// TwinCAT 3 PLC project TcKNXnetIP_Tunneling_Lib
// Title: TcKNXnetIP_Tunneling_Lib
// Company: Gauggel
// Author: Gauggel Alexander
// ProjectVersion: 1.0.0
// Description: Library for KNXnetIP Tunnelling connection (write/read group addresses) License: MIT License Disclaimer: This software is provided "as is", without warranty of any kind, express or implied. The author shall not be held liable for any damages arising from the use of this software.
// ProgramVersion: 3.1.4026.20
// libraries:
//   Tc2_Standard, * (Beckhoff Automation GmbH)
//   Tc2_System, * (Beckhoff Automation GmbH)
//   Tc2_TcpIp, * (Beckhoff Automation GmbH)
// project tree:
//   KNXnetIPTunnelingServer/DUTs/ E_KNXnetIP_COMMON_CONSTANTS.TcDUT, E_KNXnetIP_COMMON_ERROR.TcDUT, E_KNXnetIP_CONNECTIONSTATE_RESPONSE_ERROR.TcDUT, E_KNXnetIP_CONNECTION_TYPE.TcDUT, E_KNXnetIP_CONNECT_RESPONSE_ERROR.TcDUT, E_KNXnetIP_CORE.TcDUT, E_KNXnetIP_DEVICE_MANAGEMENT.TcDUT, E_KNXnetIP_ROUTING.TcDUT, E_KNXnetIP_ServiceTypes.TcDUT, E_KNXnetIP_TUNNELING.TcDUT, E_KNXnetIP_TUNNELING_CONNECT_ERROR.TcDUT, ST_KNXnetIP_cEMI.TcDUT, ST_KNXnetIP_CommonHeader.TcDUT, ST_KNXnetIP_ConnectionHeader.TcDUT, ST_KNXnetIP_ConnectionStateResponse.TcDUT, ST_KNXnetIP_ConnectResponse.TcDUT, ST_KNXnetIP_DisconnectRequest.TcDUT, ST_KNXnetIP_DisconnectResponse.TcDUT, ST_KNXnetIP_Message.TcDUT, ST_KNXnetIP_MessageOfAllGroupAddresses.TcDUT, ST_KNXnetIP_Message_Buffer.TcDUT, ST_KNX_GroupAddress.TcDUT, ST_KNX_PhysicalAddress.TcDUT
//   KNXnetIPTunnelingServer/DUTs/Interpreter/ ST_KNX_DPT_B2.TcDUT, ST_KNX_DPT_ControlDimming.TcDUT
//   KNXnetIPTunnelingServer/DUTs/StateMachines/ E_KNXnetIPStateConnection.TcDUT, E_KNXnetIPStateReceivedTelegrams.TcDUT, E_KNXnetIPStateRequest.TcDUT, E_KNXnetIPStateTransmitTelegrams.TcDUT
//   KNXnetIPTunnelingServer/ITFs/ I_KNXnetIP_Tunneling.TcIO, I_KNX_DPT_Builder.TcIO, I_KNX_DPT_Interpreter.TcIO
//   KNXnetIPTunnelingServer/PARAMs/ KNXnetIP_TIMEOUT_CONSTANS.TcGVL
//   KNXnetIPTunnelingServer/POUs/ F_KNX_GROUPADDRESS_TO_WORD.TcPOU, F_KNX_PHYSICALADDRESS_TO_WORD.TcPOU, F_WORD_TO_KNX_GROUPADDRESS.TcPOU, F_WORD_TO_KNX_PHYSICALADDRESS.TcPOU, KNXnetIPTunnelingServer.TcPOU, KNXnetIP_Message_FiFoBuffer.TcPOU, KNX_DatapointTypes_Builder.TcPOU, KNX_DatapointTypes_Interpreter.TcPOU
//   KNXnetIP_Devices/Button/ FB_KNXnetIP_Button.TcPOU
//   KNXnetIP_Devices/ FB_KNXnetIP_Device_Abstract.TcPOU
//   KNXnetIP_Devices/Light/ FB_KNXnetIP_Light.TcPOU
//   Project Information/ F_GetCompany.TcPOU, F_GetTitle.TcPOU, F_GetVersion.TcPOU
//   Version/ Global_Version.TcGVL

// ---- KNXnetIPTunnelingServer/DUTs/E_KNXnetIP_COMMON_CONSTANTS.TcDUT
{attribute 'qualified_only'}
{attribute 'to_string'}
TYPE E_KNXnetIP_COMMON_CONSTANTS :
(
	KNXNETIP_VERSION_10 := 16#10,			// Identifier for KNXnet/IP protocol version 1.0
	HEADER_SIZE_10		:= 16#06			// constant size of KNXnet/IP header as defined in protocol version 1.0
) BYTE
;
END_TYPE

// ---- KNXnetIPTunnelingServer/DUTs/E_KNXnetIP_COMMON_ERROR.TcDUT
{attribute 'qualified_only'}
{attribute 'to_string'}
TYPE E_KNXnetIP_COMMON_ERROR :
(
	E_NO_ERROR 					:= 16#00,			// Operation successful
	E_HOST_PROTOCOL_TYPE 		:= 16#01,			// The requested host protocol is not supported by the KNXnet/IP device.
	E_VERSION_NOT_SUPPORTED		:= 16#02,			// The requested protocol version is not supported by the KNXnet/IP device.
	E_SEQUENCE_NUMBER	 		:= 16#04,			// The received sequence number is out of order.
	E_ERROR 					:= 16#0F			// Any further undefined, possibly implementation specific error has occurred.
) BYTE 
;
END_TYPE

// ---- KNXnetIPTunnelingServer/DUTs/E_KNXnetIP_CONNECTIONSTATE_RESPONSE_ERROR.TcDUT
{attribute 'qualified_only'}
{attribute 'to_string'}
TYPE E_KNXnetIP_CONNECTIONSTATE_RESPONSE_ERROR :
(
	E_NO_ERROR 					:= 16#00,		// The connection state is normal.
	E_CONNECTION_ID 			:= 16#21,		// The KNXnet/IP Server device cannot find an active data connection with the specified ID.
	E_DATA_CONNECTION 			:= 16#26,		// The KNXnet/IP Server device detects an error concerning the data connection with the specified ID.
	E_KNX_CONNECTION 			:= 16#27		// The KNXnet/IP Server device detects an error concerning the KNX connection with the specified ID.
) BYTE 
;
END_TYPE

// ---- KNXnetIPTunnelingServer/DUTs/E_KNXnetIP_CONNECTION_TYPE.TcDUT
{attribute 'qualified_only'}
{attribute 'to_string'}
TYPE E_KNXnetIP_CONNECTION_TYPE :
(
	DEVICE_MGMT_CONNECTION		:= 16#03,			// Data connection used to configure a KNXnet/IP device.
	TUNNEL_CONNECTION			:= 16#04,			// Data connection used to forward KNX telegrams between two KNXnet/IP devices.
	REMLOG_CONNECTION			:= 16#06,			// Data connection used for configuration and data transfer with a remote logging server.
	REMCONF_CONNECTION			:= 16#07,			// Data connection used for data transfer with a remote configuration server.
	OBJSVR_CONNECTION			:= 16#08			// Data connection used for configuration and data transfer with an Object Server in a KNXnet/IP device. 
) BYTE
;
END_TYPE

// ---- KNXnetIPTunnelingServer/DUTs/E_KNXnetIP_CONNECT_RESPONSE_ERROR.TcDUT
{attribute 'qualified_only'}
{attribute 'to_string'}
TYPE E_KNXnetIP_CONNECT_RESPONSE_ERROR :
(
	E_NO_ERROR 						:= 16#00,		// The connection is established successfully.
	E_CONNECTION_TYPE 				:= 16#22,		// The KNXnet/IP Server device does not support the requested connection type.
	E_CONNECTION_OPTION 			:= 16#23,		// The KNXnet/IP Server device does not support one or more requested connection options.
	E_NO_MORE_CONNECTIONS 			:= 16#24,		// The KNXnet/IP Server device cannot accept the new data connection because its maximum amount of concurrent connections is already used.
	E_AUTHORISATION_ERROR 			:= 16#28,		// The Client is not authorised to establish the requested connection The Client is not authorised to use the requested IA in the Extended CRI.
	E_NO_TUNNELING_ADDRESS 			:= 16#2D,		// The IA requested in the Extended CRI is not a Tunnelling IA.
	E_CONNECTION_IN_USE 			:= 16#2E		// The IA requested for this connection is in use. 
) BYTE
;
END_TYPE

// ---- KNXnetIPTunnelingServer/DUTs/E_KNXnetIP_CORE.TcDUT
{attribute 'qualified_only'}
{attribute 'to_string'}
TYPE E_KNXnetIP_CORE :
(
	SEARCH_REQUEST 				:= 16#0201,		// Sent by KNXnet/IP Client to search available KNXnet/IP Servers
	SEARCH_RESPONSE				:= 16#0202,		// Sent by KNXnet/IP Server when receiving a KNXnet/IP SEARCH_REQUEST
	DESCRIPITON_REQUEST			:= 16#0203,		// Sent by KNXnet/IP Client to a KNXnet/IP Server to retrieve information about capabilities and supported services
	DESCRIPTION_RESPONSE		:= 16#0204,		// Sent by KNXnet/IP Server in response to a DESCRIPTION_REQUEST to provide information about the server implementation
	CONNECT_REQUEST				:= 16#0205,		// Sent by KNXnet/IP Client for establishing a communication channel to a KNXnet/IP Server.
	CONNECT_RESPONSE			:= 16#0206,		// Sent by KNXnet/IP Server as answer to CONNECT_REQUEST telegram.
	CONNECTIONSTATE_REQUEST		:= 16#0207,		// Sent by KNXnet/IP Client for requesting the connection state of an established connection to a KNXnet/IP Server.
	CONNECTIONSTATE_RESPONSE	:= 16#0208,		// Sent by KNXnet/IP Server when receiving a CONNECTIONSTATE_REQUEST for an established connection.
	DISCONNECT_REQUEST			:= 16#0209,		// Sent by KNXnet/IP device, typically the KNXnet/IP Client, to terminate an established connection.
	DISCONNECT_RESPONSE			:= 16#020A,		// Sent by KNXnet/IP device, typically the KNXnet/IP Server, in response to a DISCONNECT_REQUEST.
	SECURE_WRAPPER				:= 16#0950,		// Contains an encrypted frame plus data for ensuring data integrity and freshness.
	SESSION_REQUEST				:= 16#0951,		// Used to initiate the secure connection setup handshake for a new secure communication session.
	SESSION_RESPONSE			:= 16#0952,		// Sent in response to a received secure session request frame.
	SESSION_AUTHENTICATE		:= 16#0953,		// Sent after the Diffie-Hellman handshake to authenticate the user against the server.
	SESSION_STATUS				:= 16#0954,		// Sent in any stage of the secure session handshake to indicate an error condition or status information.
	TIMER_NOTIFY				:= 16#0955		// Used to ensure synchronization of the multicast group member's timer values.
) WORD 
;
END_TYPE

// ---- KNXnetIPTunnelingServer/DUTs/E_KNXnetIP_DEVICE_MANAGEMENT.TcDUT
{attribute 'qualified_only'}
{attribute 'to_string'}
TYPE E_KNXnetIP_DEVICE_MANAGEMENT :
(
	DEVICE_CONFIGURATION_REQUEST	:= 16#0310,			// Reads/Writes KNXnet/IP device configuration data (Interface Object Properties)
	DEVICE_CONFIGURATION_ACK		:= 16#0311			// Sent by a KNXnet/IP device to confirm the reception of the DEVICE_CONFIGURATION_REQUEST. 
) WORD 
;
END_TYPE

// ---- KNXnetIPTunnelingServer/DUTs/E_KNXnetIP_ROUTING.TcDUT
{attribute 'qualified_only'}
{attribute 'to_string'}
TYPE E_KNXnetIP_ROUTING :
(
	ROUTING_INDICATION 		:= 16#0530,		// Used for sending KNX telegrams over IP networks. This service is unconfirmed.
	ROUTING_LOST_MESSAGE	:= 16#0531		// Used for indication of lost KNXnet/IP Routing messages. This service is unconfirmed.
) WORD
;
END_TYPE

// ---- KNXnetIPTunnelingServer/DUTs/E_KNXnetIP_ServiceTypes.TcDUT
{attribute 'qualified_only'}
{attribute 'to_string'}
TYPE E_KNXnetIP_ServiceTypes :
(
	eL_DataReq		 	:= 16#11,
	eL_DataCon			:= 16#2E,
	eL_DataInd			:= 16#29
)BYTE
;
END_TYPE

// ---- KNXnetIPTunnelingServer/DUTs/E_KNXnetIP_TUNNELING.TcDUT
{attribute 'qualified_only'}
{attribute 'to_string'}
TYPE E_KNXnetIP_TUNNELING :
(
	TUNNELING_REQUEST 	:= 16#0420,		// Used for sending and receiving single KNX telegrams between KNXnet/IP Client and - Server.
	TUNNELING_ACK		:= 16#0421		// Sent by a KNXnet/IP device to confirm the reception of the TUNNELING_REQUEST.
) WORD
;
END_TYPE

// ---- KNXnetIPTunnelingServer/DUTs/E_KNXnetIP_TUNNELING_CONNECT_ERROR.TcDUT
{attribute 'qualified_only'}
{attribute 'to_string'}
TYPE E_KNXnetIP_TUNNELING_CONNECT_ERROR :
(
	E_NO_ERROR			:= 16#00,		// The message is received successfully.
	E_TUNNELING_LAYER	:= 16#29		// The KNXnet/IP Server device does not support the requested KNXnet/IP Tunneling layer.
) BYTE
;
END_TYPE

// ---- KNXnetIPTunnelingServer/DUTs/Interpreter/ST_KNX_DPT_B2.TcDUT
TYPE ST_KNX_DPT_B2 :
STRUCT
	bBit1			: BOOL;
	bBit2			: BOOL;
END_STRUCT
END_TYPE

// ---- KNXnetIPTunnelingServer/DUTs/Interpreter/ST_KNX_DPT_ControlDimming.TcDUT
TYPE ST_KNX_DPT_ControlDimming :
STRUCT
	bControl		: BOOL;		// 0 = Decrease, 1 = Increase
	nStepCode		: BYTE;		// 001b..111b: Step number of intervals = 2^(stepcode-1); 000b: Break
END_STRUCT
END_TYPE

// ---- KNXnetIPTunnelingServer/DUTs/StateMachines/E_KNXnetIPStateConnection.TcDUT
{attribute 'qualified_only'}
{attribute 'strict'}
{attribute 'to_string'}
TYPE E_KNXnetIPStateConnection :
(
	eInit 									:= 0,
	eDisconnected							:= 1,
	eCreateUdpSocket						:= 2,
	eSendConnectRequestToTunnelingServer	:= 3,
	eWaitForConnectResponse					:= 4,
	eConnected								:= 5,
	eSendConnectionStateRequest				:= 6,
	eWaitForConnectionStateResponse			:= 7,
	eDisconnectValidConnection				:= 10,
	eWaitForDisconnectResponse				:= 11,
	eAckDisconnectReq						:= 98,
	eCloseAllSockets						:= 99,
	eError									:= 100
);
END_TYPE

// ---- KNXnetIPTunnelingServer/DUTs/StateMachines/E_KNXnetIPStateReceivedTelegrams.TcDUT
{attribute 'qualified_only'}
{attribute 'strict'}
{attribute 'to_string'}
TYPE E_KNXnetIPStateReceivedTelegrams :
(
	eInit 									:= 0,
	eWaitForNextTelegram					:= 1
);
END_TYPE

// ---- KNXnetIPTunnelingServer/DUTs/StateMachines/E_KNXnetIPStateRequest.TcDUT
{attribute 'qualified_only'}
{attribute 'strict'}
{attribute 'to_string'}
TYPE E_KNXnetIPStateRequest :
(
	eInit 									:= 0,
	eWaitForNextRequest						:= 1
);
END_TYPE

// ---- KNXnetIPTunnelingServer/DUTs/StateMachines/E_KNXnetIPStateTransmitTelegrams.TcDUT
{attribute 'qualified_only'}
{attribute 'strict'}
{attribute 'to_string'}
TYPE E_KNXnetIPStateTransmitTelegrams :
(
	eInit 									:= 0,
	eWaitForNextTelegramToTransmit			:= 1,
	eTransmit								:= 2,
	eWaitTimeForNextTransmit				:= 3
);
END_TYPE

// ---- KNXnetIPTunnelingServer/DUTs/ST_KNXnetIP_cEMI.TcDUT
TYPE ST_KNXnetIP_cEMI :
STRUCT
	nMessageCode				: BYTE;
	nAdditionalInfoLength		: BYTE;
	nAdditionalInfo				: ARRAY[0..20] OF BYTE;
	nControlField1				: BYTE;
	nControlField2				: BYTE;
	nSourcePhysicalAddress		: WORD;
	stSourcePhysicalAddress		: ST_KNX_PhysicalAddress;
	nDestinationGroupAddress	: WORD;
	stDestinationGroupAddress	: ST_KNX_GroupAddress;
	LengthDataField				: BYTE;
	Data						: ARRAY[1..255] OF BYTE;
END_STRUCT
END_TYPE

// ---- KNXnetIPTunnelingServer/DUTs/ST_KNXnetIP_CommonHeader.TcDUT
TYPE ST_KNXnetIP_CommonHeader :
STRUCT
	nHeaderSize			: BYTE;
	nProtocolVersion	: BYTE;
	nServiceType		: WORD;
	nTotalLength		: WORD;
END_STRUCT
END_TYPE

// ---- KNXnetIPTunnelingServer/DUTs/ST_KNXnetIP_ConnectionHeader.TcDUT
TYPE ST_KNXnetIP_ConnectionHeader :
STRUCT
	nStructureLength			: BYTE;
	nCommunicationChannel		: BYTE;
	nSequenceCounter			: BYTE;
	nReserved					: BYTE;
END_STRUCT
END_TYPE

// ---- KNXnetIPTunnelingServer/DUTs/ST_KNXnetIP_ConnectionStateResponse.TcDUT
TYPE ST_KNXnetIP_ConnectionStateResponse EXTENDS ST_KNXnetIP_CommonHeader :
STRUCT
	nCommunicationChannelID		: BYTE;
	nStatusCode					: E_KNXnetIP_CONNECTIONSTATE_RESPONSE_ERROR;
END_STRUCT
END_TYPE

// ---- KNXnetIPTunnelingServer/DUTs/ST_KNXnetIP_ConnectResponse.TcDUT
TYPE ST_KNXnetIP_ConnectResponse EXTENDS ST_KNXnetIP_CommonHeader :
STRUCT
	nCommunicationChannelID		: BYTE;
	nStatusCode					: E_KNXnetIP_CONNECT_RESPONSE_ERROR;
	nStructureLength			: BYTE;
	nHostProtocolCode			: BYTE;
	nDataEndpointIPv4			: DWORD;
	nDataEndpointPort			: WORD;
	nStructueLengthCRD			: BYTE;
	nConnectionTypeCode			: BYTE;
	nPhysicalAddress			: WORD;
END_STRUCT
END_TYPE

// ---- KNXnetIPTunnelingServer/DUTs/ST_KNXnetIP_DisconnectRequest.TcDUT
TYPE ST_KNXnetIP_DisconnectRequest EXTENDS ST_KNXnetIP_CommonHeader :
STRUCT
	nCommunicationChannelID		: BYTE;
	nStructLength				: BYTE;	
	nHostProtocolCode			: BYTE;
	nControlEndpointIPv4		: DWORD;
	nControlEndpointPort		: WORD;
END_STRUCT
END_TYPE

// ---- KNXnetIPTunnelingServer/DUTs/ST_KNXnetIP_DisconnectResponse.TcDUT
TYPE ST_KNXnetIP_DisconnectResponse EXTENDS ST_KNXnetIP_CommonHeader :
STRUCT
	nCommunicationChannelID		: BYTE;
	nStatusCode					: E_KNXnetIP_CONNECT_RESPONSE_ERROR;
END_STRUCT
END_TYPE

// ---- KNXnetIPTunnelingServer/DUTs/ST_KNXnetIP_Message.TcDUT
TYPE ST_KNXnetIP_Message :
STRUCT
	aMessage		: ARRAY[1..255] OF BYTE;		// byte array of message
	nByteLength		: UDINT := SIZEOF(aMessage);	// count of used bytes for message
END_STRUCT
END_TYPE

// ---- KNXnetIPTunnelingServer/DUTs/ST_KNXnetIP_MessageOfAllGroupAddresses.TcDUT
TYPE ST_KNXnetIP_MessageOfAllGroupAddresses :
STRUCT
	aMessage		: ARRAY[0..31, 0..7, 0..255] OF ARRAY[1..255] OF BYTE;
	aTimeStamp		: ARRAY[0..31, 0..7, 0..255] OF DT;
	aNewMessage		: ARRAY[0..31, 0..7, 0..255] OF BOOL;
END_STRUCT
END_TYPE

// ---- KNXnetIPTunnelingServer/DUTs/ST_KNXnetIP_Message_Buffer.TcDUT
TYPE ST_KNXnetIP_Message_Buffer :
STRUCT
	aKNXnetIP_Messages		: ARRAY[1..255] OF ST_KNXnetIP_Message;		// array of messages
END_STRUCT
END_TYPE

// ---- KNXnetIPTunnelingServer/DUTs/ST_KNX_GroupAddress.TcDUT
TYPE ST_KNX_GroupAddress :
STRUCT
	nFirst			: UINT;			// first number of group address 1/x/x
	nMiddle			: UINT;			// second number of group address x/1/x
	nLow			: UINT;			// third number of group address x/x/1
END_STRUCT
END_TYPE

// ---- KNXnetIPTunnelingServer/DUTs/ST_KNX_PhysicalAddress.TcDUT
TYPE ST_KNX_PhysicalAddress :
STRUCT
	nArea		: BYTE;			// first number of physical address 1.x.x
	nLine		: BYTE;			// second number of physical address x.1.x
	nDevice		: BYTE;			// third number of physical address x.x.1
END_STRUCT
END_TYPE

// ---- KNXnetIPTunnelingServer/PARAMs/KNXnetIP_TIMEOUT_CONSTANS.TcGVL
VAR_GLOBAL CONSTANT
	CONNECT_REQUEST_TIMEOUT					: TIME := T#10S;		// KNXnet/IP Client shall wait for 10 seconds for a CONNECT_RESPONSE frame from KNXnet/IP Server.
	CONNECTIONSTATE_REQUEST_TIMEOUT			: TIME := T#10S;		// KNXnet/IP Client shall wait for 10 seconds for a CONNECTIONSTATE_RESPONSE frame from KNXnet/IP Server.
	DEVICE_CONFIGURATION_REQUEST_TIMEOUT	: TIME := T#10S;		// KNXnet/IP Client shall wait for 10 seconds for a DEVICE_CONFIGURATION_RESPONSE frame from KNXnet/IP Server.
	TUNNELING_REQUEST_TIMEOUT				: TIME := T#1S;			// KNXnet/IP Client shall wait for 1 second for a TUNNELING_ACK response on a TUNNELING_REQUEST frame from KNXnet/IP Server.
	CONNECTION_ALIVE_TIME					: TIME := T#120S;		// If the KNXnet/IP Server does not receive a heartbeat request within 120 seconds of the last correctly received message frame, the server shall terminate the connection by sending a DISCONNECT_REQUEST to the client’s control endpoint.
	CONNECTION_HEARTBEAT_TIME				: TIME := T#40S;		// heartbeat time to send a new connection state request
END_VAR

// ---- Version/Global_Version.TcGVL
{attribute 'TcGenerated'}
{attribute 'no-analysis'}
{attribute 'linkalways'}
// This function has been automatically generated from the project information.
VAR_GLOBAL CONSTANT
	{attribute 'const_non_replaced'}
	stLibVersion_TcKNXnetIP_Tunneling_Lib : ST_LibVersion := (iMajor := 1, iMinor := 0, iBuild := 0, iRevision := 0, nFlags := 1, sVersion := '1.0.0');
END_VAR

// ---- KNXnetIPTunnelingServer/ITFs/I_KNXnetIP_Tunneling.TcIO
INTERFACE I_KNXnetIP_Tunneling

(* 
	transmitting group address message to tunneling server
*)
METHOD M_TransmitMessage : BOOL
VAR_INPUT
	stInGroupAddress		: ST_KNX_GroupAddress;			// group address
	stInMessage				: ST_KNXnetIP_Message;			// message to send
END_VAR
END_METHOD

(*
	return reference to the messages of all group addresses
*)
PROPERTY P_G_GroupAddressMessages : REFERENCE TO ST_KNXnetIP_MessageOfAllGroupAddresses
GET
END_GET
END_PROPERTY

(*
	host has valid connection to tunneling server
*)
PROPERTY P_G_IsConnected : BOOL
GET
END_GET
END_PROPERTY

(*
	physical address of host
*)
PROPERTY P_G_PhysicalAddress : REFERENCE TO ST_KNX_PhysicalAddress
GET
END_GET
END_PROPERTY

END_INTERFACE

// ---- KNXnetIPTunnelingServer/ITFs/I_KNX_DPT_Builder.TcIO
INTERFACE I_KNX_DPT_Builder

METHOD M_Build2Bit : ST_KNXnetIP_Message
VAR_INPUT
	bInValueBit1	: BOOL;
	bInValueBit2	: BOOL;
END_VAR
END_METHOD

METHOD M_Build3Byte : ST_KNXnetIP_Message
VAR_INPUT
	nInValue		: DWORD;
END_VAR
END_METHOD

METHOD M_BuildBool : ST_KNXnetIP_Message
VAR_INPUT
	bInValue	: BOOL;
END_VAR
END_METHOD

METHOD M_BuildDimming : ST_KNXnetIP_Message
VAR_INPUT
	stInValue		: ST_KNX_DPT_ControlDimming;
END_VAR
END_METHOD

METHOD M_BuildFloat16 : ST_KNXnetIP_Message
VAR_INPUT
	fInValue	: REAL;
END_VAR
END_METHOD

METHOD M_BuildINT16 : ST_KNXnetIP_Message
VAR_INPUT
	nInValue	: INT;
END_VAR
END_METHOD

METHOD M_BuildINT32 : ST_KNXnetIP_Message
VAR_INPUT
	nInValue	: DINT;
END_VAR
END_METHOD

METHOD M_BuildString : ST_KNXnetIP_Message
VAR_INPUT
	sInValue	: STRING;
END_VAR
END_METHOD

METHOD M_BuildUINT16 : ST_KNXnetIP_Message
VAR_INPUT
	nInValue	: UINT;
END_VAR
END_METHOD

METHOD M_BuildUINT32 : ST_KNXnetIP_Message
VAR_INPUT
	nInValue	: UDINT;
END_VAR
END_METHOD

METHOD M_BuildUINT8 : ST_KNXnetIP_Message
VAR_INPUT
	nInValue		: BYTE;
END_VAR
END_METHOD

END_INTERFACE

// ---- KNXnetIPTunnelingServer/ITFs/I_KNX_DPT_Interpreter.TcIO
INTERFACE I_KNX_DPT_Interpreter

METHOD M_InterpretAs2Bit : ST_KNX_DPT_B2
VAR_IN_OUT
	aInData		: ARRAY[*] OF BYTE;
END_VAR
END_METHOD

METHOD M_InterpretAsBool : BOOL
VAR_IN_OUT
	aInData		: ARRAY[*] OF BYTE;
END_VAR
END_METHOD

METHOD M_InterpretAsDimming : ST_KNX_DPT_ControlDimming
VAR_IN_OUT
	aInData		: ARRAY[*] OF BYTE;
END_VAR
END_METHOD

METHOD M_InterpretAsFloat16 : REAL
VAR_IN_OUT
	aInData		: ARRAY[*] OF BYTE;
END_VAR
END_METHOD

METHOD M_InterpretAsFloat32 : Real
VAR_IN_OUT
	aInData		: ARRAY[*] OF BYTE;
END_VAR
END_METHOD

METHOD M_InterpretAsINT16 : INT
VAR_IN_OUT
	aInData		: ARRAY[*] OF BYTE;
END_VAR
END_METHOD

METHOD M_InterpretAsINT32 : DINT
VAR_IN_OUT
	aInData		: ARRAY[*] OF BYTE;
END_VAR
END_METHOD

METHOD M_InterpretAsUINT16 : UINT
VAR_IN_OUT
	aInData		: ARRAY[*] OF BYTE;
END_VAR
END_METHOD

METHOD M_InterpretAsUINT32 : UDINT
VAR_IN_OUT
	aInData		: ARRAY[*] OF BYTE;
END_VAR
END_METHOD

METHOD M_InterpretAsUINT8 : BYTE
VAR_IN_OUT
	aInData		: ARRAY[*] OF BYTE;
END_VAR
END_METHOD

METHOD M_InterpretNewMessage : BOOL
VAR_IN_OUT
	bInData		: BOOL;
END_VAR
END_METHOD

END_INTERFACE

// ---- KNXnetIPTunnelingServer/POUs/F_KNX_GROUPADDRESS_TO_WORD.TcPOU
FUNCTION F_KNX_GROUPADDRESS_TO_WORD : WORD
VAR_INPUT
	stInGroupAddress		: ST_KNX_GroupAddress;
END_VAR
VAR
	nResult				: WORD;
END_VAR

nResult		:= SHL(UINT_TO_WORD(stInGroupAddress.nFirst), 11);
nResult		:= nResult OR SHL(UINT_TO_WORD(stInGroupAddress.nMiddle), 8);
nResult 	:= nResult OR UINT_TO_WORD(stInGroupAddress.nLow);
F_KNX_GROUPADDRESS_TO_WORD := nResult;

END_FUNCTION

// ---- KNXnetIPTunnelingServer/POUs/F_KNX_PHYSICALADDRESS_TO_WORD.TcPOU
FUNCTION F_KNX_PHYSICALADDRESS_TO_WORD : WORD
VAR_INPUT
	stInPhysicalAddress		: ST_KNX_PhysicalAddress;
END_VAR
VAR
	nResult					: WORD;
END_VAR

nResult			:= SHL(BYTE_TO_WORD(stInPhysicalAddress.nArea), 4*3);
nResult			:= nResult OR SHL(BYTE_TO_WORD(stInPhysicalAddress.nLine),4*2);
nResult			:= nResult OR BYTE_TO_WORD(stInPhysicalAddress.nDevice);
F_KNX_PHYSICALADDRESS_TO_WORD := nResult;

END_FUNCTION

// ---- KNXnetIPTunnelingServer/POUs/F_WORD_TO_KNX_GROUPADDRESS.TcPOU
FUNCTION F_WORD_TO_KNX_GROUPADDRESS : ST_KNX_GroupAddress
VAR_INPUT
	nInGroupAddress			: WORD;
END_VAR
VAR
	stResult				: ST_KNX_GroupAddress;
END_VAR

stResult.nFirst		:= SHR(nInGroupAddress AND 16#F800, 11);
stResult.nMiddle	:= SHR(nInGroupAddress AND 16#0700, 8);
stResult.nLow		:= nInGroupAddress AND 16#FF;
F_WORD_TO_KNX_GROUPADDRESS := stResult;

END_FUNCTION

// ---- KNXnetIPTunnelingServer/POUs/F_WORD_TO_KNX_PHYSICALADDRESS.TcPOU
FUNCTION F_WORD_TO_KNX_PHYSICALADDRESS : ST_KNX_PhysicalAddress
VAR_INPUT
	nInPhysicalAddress		: WORD;
END_VAR
VAR
	stResult				: ST_KNX_PhysicalAddress;
END_VAR

stResult.nArea		:= WORD_TO_BYTE(SHR(nInPhysicalAddress AND 16#F000, 4*3));
stResult.nLine		:= WORD_TO_BYTE(SHR(nInPhysicalAddress AND 16#0F00, 4*2));
stResult.nDevice	:= WORD_TO_BYTE(nInPhysicalAddress AND 16#00FF);
F_WORD_TO_KNX_PHYSICALADDRESS := stResult;

END_FUNCTION

// ---- KNXnetIPTunnelingServer/POUs/KNXnetIPTunnelingServer.TcPOU
(*
:Description: This function block is the heart of the library. It will connecting to the tunnelling server and send/receive telegrams.
:Instructions for use: For every tunneling server you have to declare this fb. It is possible to use more tunneling at the same time with different physical addresses (the tunneling server should have more than one available server).
*)
FUNCTION_BLOCK KNXnetIPTunnelingServer IMPLEMENTS I_KNXnetIP_Tunneling
VAR_INPUT
	stInPhysicalAddress					: ST_KNX_PhysicalAddress;						// physical address of local host, mostly needed to see in ETS the local host device
	sInSrvNetId							: T_AmsNetID 	:= '';							// net-id of twincat system, if local than use empty string ''
	sInLocalHostIPv4Addr				: T_IPv4Addr;									// ipv4 address of the local host
	nInLocalPort						: UINT;											// port for communication on local host
	                            		                            					
	sInRemoteHostIPv4Addr				: T_IPv4Addr;									// ipv4 address of the remote host, which should be connected
	nInRemotePort						: UINT;											// port for communication on remote host
	DateAndTime							: DT;											// Actuall Date and Time for Timestamp
END_VAR             		                                        		
VAR                             		                                        		
	bInit								: BOOL := FALSE;	                    		
                                		                                        		
	bInitiateConnection					: BOOL;											// initiation of the connection
	bInitiateDisconnection				: BOOL;											// initiation of disconnect the connection
	                            		                                        		
	// receive                  		                                        		
	fbReceiveFiFoBuffer					: KNXnetIP_Message_FiFoBuffer;					// receive fifo buffer for KNXnetIP messages
	                            	                                            		
	// transmit                 	                                            		
	fbTransmitFiFoBuffer				: KNXnetIP_Message_FiFoBuffer;					// transmit fifo buffer for KNXnetIP messages
	fbTransmitFiFoBufferQuick			: KNXnetIP_Message_FiFoBuffer;					// transmit quick fifo buffer for KNXnetIP messages
	                                                                            		
	// important communication variables                                        	
	nCommunicationChannelID				: BYTE;											// communication channel ID for further communications, is received from server
	nPhysicalAddressTunneling			: WORD;											// physical address to comunicate over tunneling server, is received from server
	
	// backing
	_bIsConnected						: BOOL;
	_bIsConnecting						: BOOL;
	_bIsDisconnecting					: BOOL;
	_bDisconnectReceived				: BOOL;
	_bTunnelReqReceived					: BOOL;
	_bTunnellingAckReceived				: BOOL;
	_bConnectionStateResponseReceived	: BOOL;
	_bConnectResponseReceived			: BOOL;
	_bDisconnectResponseReceived		: BOOL;
	_bReconnect							: BOOL;
	_bTransmitTimeout					: BOOL;
	_nSequenceCounter					: BYTE := 255;
	_nSequenceCounterTransmit			: BYTE := 0;
	_stConnectedSocket					: T_HSOCKET;									// actually connected socket
	_stPhysicalAddressTunneling			: ST_KNX_PhysicalAddress;						// physical Address for tunneling server, which is got from server at connect request
	
END_VAR
VAR_STAT 
	stGroupAddressMessages				: ST_KNXnetIP_MessageOfAllGroupAddresses;		// reference to all group addresses, for writing
END_VAR

IF bInit THEN
	M_Init();
END_IF

M_ManagerTransmit();
M_ManagerConnection();
M_ManagerReceiving();
M_ManagerConvertReceived();

METHOD PRIVATE M_AddHPAI : BOOL
VAR_IN_OUT
	stInMessage					: ST_KNXnetIP_Message;		// message to add the HPAI
END_VAR
VAR_INPUT	
	nInStartByte				: UINT;						// starting byte, where the HPAI should be added
	sInIPv4Addr					: T_IPv4Addr;				// ipv4 address of HPAI
	nInPortNumber				: UINT;						// port number of HPAI
END_VAR	
VAR
	aIPv4Address				: T_IPv4AddrArr;			// ipv4 address in bytes
END_VAR
VAR CONSTANT
	cStructLengthHPAI			: BYTE := 16#08;			// structure length of HPAI are 8 octetts
	cIPV4_UDP					: BYTE := 16#01;			// identifier for protocol version 4 address and port number for UDP communication
END_VAR
// insert HPAI at start byte position
stInMessage.aMessage[nInStartByte] 		:= cStructLengthHPAI;
stInMessage.aMessage[nInStartByte+1] 	:= cIPV4_UDP;
aIPv4Address							:= F_ScanIPv4AddrIds(sInIPv4Addr);
stInMessage.aMessage[nInStartByte+2] 	:= aIPv4Address[0];
stInMessage.aMessage[nInStartByte+3] 	:= aIPv4Address[1];
stInMessage.aMessage[nInStartByte+4] 	:= aIPv4Address[2];
stInMessage.aMessage[nInStartByte+5] 	:= aIPv4Address[3];
stInMessage.aMessage[nInStartByte+6] 	:= M_GetHighByte(UINT_TO_WORD(nInPortNumber));
stInMessage.aMessage[nInStartByte+7] 	:= M_GetLowByte(UINT_TO_WORD(nInPortNumber));
END_METHOD

METHOD PRIVATE M_AreHostAndPortValid : BOOL
VAR_INPUT	
	sHost						: T_IPv4Addr;						// host, which are the data was received
	nPort						: UDINT;							// port, which are the data was received
END_VAR
M_AreHostAndPortValid := (sHost = sInRemoteHostIPv4Addr) AND (nPort = nInRemotePort);
END_METHOD

METHOD PRIVATE M_BuildDisconnectResponse : ST_KNXnetIP_Message
VAR
	stResult			: ST_KNXnetIP_Message;
	aIPv4Address		: T_IPv4AddrArr;			// ipv4 address in bytes
END_VAR
VAR CONSTANT
	cTotalLength		: WORD := 16#0008;			// total length ares 8 octetts
END_VAR
// ------ KNXnet/IP header
stResult.aMessage[1] 	:= E_KNXnetIP_COMMON_CONSTANTS.HEADER_SIZE_10;
stResult.aMessage[2] 	:= E_KNXnetIP_COMMON_CONSTANTS.KNXNETIP_VERSION_10;
stResult.aMessage[3] 	:= M_GetHighByte(E_KNXnetIP_CORE.DISCONNECT_RESPONSE);
stResult.aMessage[4] 	:= M_GetLowByte(E_KNXnetIP_CORE.DISCONNECT_RESPONSE);
stResult.aMessage[5] 	:= M_GetHighByte(cTotalLength);
stResult.aMessage[6] 	:= M_GetLowByte(cTotalLength);
stResult.aMessage[7]	:= nCommunicationChannelID;
stResult.aMessage[8]	:= E_KNXnetIP_CONNECTIONSTATE_RESPONSE_ERROR.E_NO_ERROR;

// set length
stResult.nByteLength := WORD_TO_UINT(cTotalLength);

// return result
M_BuildDisconnectResponse := stResult;
END_METHOD

METHOD PRIVATE M_BuildTunnelConnectionStateRequest : ST_KNXnetIP_Message
VAR
	stResult			: ST_KNXnetIP_Message;
END_VAR
VAR CONSTANT
	cTotalLength		: WORD := 16#0010;			// total length ares 16 octetts
	cStructLengthHPAI	: BYTE := 16#08;			// structure length of HPAI are 8 octetts
	cIPV4_UDP			: BYTE := 16#01;			// identifier for protocol version 4 address and port number for UDP communication
	aIPv4Address		: T_IPv4AddrArr;			// ipv4 address in bytes
END_VAR
// ------ KNXnet/IP header
stResult.aMessage[1] 	:= E_KNXnetIP_COMMON_CONSTANTS.HEADER_SIZE_10;
stResult.aMessage[2] 	:= E_KNXnetIP_COMMON_CONSTANTS.KNXNETIP_VERSION_10;
stResult.aMessage[3] 	:= M_GetHighByte(E_KNXnetIP_CORE.CONNECTIONSTATE_REQUEST);
stResult.aMessage[4] 	:= M_GetLowByte(E_KNXnetIP_CORE.CONNECTIONSTATE_REQUEST);
stResult.aMessage[5] 	:= M_GetHighByte(cTotalLength);
stResult.aMessage[6] 	:= M_GetLowByte(cTotalLength);

// ------ KNXnet/IP body
// --------- Communication Channel ID
stResult.aMessage[7] 	:= nCommunicationChannelID;
stResult.aMessage[8] 	:= 16#0;	// reserved

// --------- HPAI of Client (control endpoint)
M_AddHPAI(	stInMessage 			:= stResult,
			nInStartByte			:= 9,
			sInIPv4Addr				:= sInLocalHostIPv4Addr,
			nInPortNumber			:= nInLocalPort);

// set length
stResult.nByteLength := WORD_TO_UINT(cTotalLength);

// return result
M_BuildTunnelConnectionStateRequest := stResult;
END_METHOD

METHOD PRIVATE M_BuildTunnelConnectRequest : ST_KNXnetIP_Message
VAR
	stResult			: ST_KNXnetIP_Message;
	aIPv4Address		: T_IPv4AddrArr;			// ipv4 address in bytes
END_VAR
VAR CONSTANT
	cTotalLength		: WORD := 16#001A;			// total length ares 26 octetts
	cStructLengthHPAI	: BYTE := 16#08;			// structure length of HPAI are 8 octetts
	cStructLengthCRI	: BYTE := 16#04;			// structure length of CRI are 4 octetts
	cIPV4_UDP			: BYTE := 16#01;			// identifier for protocol version 4 address and port number for UDP communication
	cTUNNEL_LINKLAYER	: BYTE := 16#02;			// KNX Layer, e.g., TUNNEL_LINKLAYER
END_VAR
// ------ KNXnet/IP header
stResult.aMessage[1] 	:= E_KNXnetIP_COMMON_CONSTANTS.HEADER_SIZE_10;
stResult.aMessage[2] 	:= E_KNXnetIP_COMMON_CONSTANTS.KNXNETIP_VERSION_10;
stResult.aMessage[3] 	:= M_GetHighByte(E_KNXnetIP_CORE.CONNECT_REQUEST);
stResult.aMessage[4] 	:= M_GetLowByte(E_KNXnetIP_CORE.CONNECT_REQUEST);
stResult.aMessage[5] 	:= M_GetHighByte(cTotalLength);
stResult.aMessage[6] 	:= M_GetLowByte(cTotalLength);

// ------ KNXnet/IP body
// --------- HPAI of Client (control endpoint)
M_AddHPAI(	stInMessage 			:= stResult,
			nInStartByte			:= 7,
			sInIPv4Addr				:= sInLocalHostIPv4Addr,
			nInPortNumber			:= nInLocalPort);

// --------- HPAI of Server (data endpoint)
M_AddHPAI(	stInMessage 			:= stResult,
			nInStartByte			:= 15,
			sInIPv4Addr				:= sInLocalHostIPv4Addr,
			nInPortNumber			:= nInLocalPort);

// --------- CRI (Connection request information)
stResult.aMessage[23] 	:= cStructLengthCRI;
stResult.aMessage[24] 	:= E_KNXnetIP_CONNECTION_TYPE.TUNNEL_CONNECTION;
stResult.aMessage[25] 	:= cTUNNEL_LINKLAYER;
stResult.aMessage[26] 	:= 16#0;	// reserved


// set length
stResult.nByteLength := WORD_TO_UINT(cTotalLength);

// return result
M_BuildTunnelConnectRequest := stResult;
END_METHOD

METHOD PRIVATE M_BuildTunnelDisconnectRequest : ST_KNXnetIP_Message
VAR
	stResult			: ST_KNXnetIP_Message;
END_VAR
VAR CONSTANT
	cTotalLength		: WORD := 16#0010;			// total length ares 16 octetts
	cStructLengthHPAI	: BYTE := 16#08;			// structure length of HPAI are 8 octetts
	cIPV4_UDP			: BYTE := 16#01;			// identifier for protocol version 4 address and port number for UDP communication
	aIPv4Address		: T_IPv4AddrArr;			// ipv4 address in bytes
END_VAR
IF NOT P_G_IsConnected THEN
	RETURN;		// no necessary connection data available!
END_IF

// ------ KNXnet/IP header
stResult.aMessage[1] 	:= E_KNXnetIP_COMMON_CONSTANTS.HEADER_SIZE_10;
stResult.aMessage[2] 	:= E_KNXnetIP_COMMON_CONSTANTS.KNXNETIP_VERSION_10;
stResult.aMessage[3] 	:= M_GetHighByte(E_KNXnetIP_CORE.DISCONNECT_REQUEST);
stResult.aMessage[4] 	:= M_GetLowByte(E_KNXnetIP_CORE.DISCONNECT_REQUEST);
stResult.aMessage[5] 	:= M_GetHighByte(cTotalLength);
stResult.aMessage[6] 	:= M_GetLowByte(cTotalLength);

// ------ KNXnet/IP body
// --------- Communication Channel ID
stResult.aMessage[7] 	:= nCommunicationChannelID;
stResult.aMessage[8] 	:= 16#0;	// reserved

// --------- HPAI of Client (control endpoint)
M_AddHPAI(	stInMessage 			:= stResult,
			nInStartByte			:= 9,
			sInIPv4Addr	:= sInLocalHostIPv4Addr,
			nInPortNumber			:= nInLocalPort);

// set length
stResult.nByteLength := WORD_TO_UINT(cTotalLength);

// return result
M_BuildTunnelDisconnectRequest := stResult;
END_METHOD

METHOD PRIVATE M_BuildTunnellingAck : ST_KNXnetIP_Message
VAR
	stResult			: ST_KNXnetIP_Message;
END_VAR
VAR CONSTANT
	cTotalLength					: WORD := 16#000A;			// total length ares 10 octetts
	cStructLengthCONNECTIONHEADER	: BYTE := 16#04;			// structure length of Connection header are 4 octetts
END_VAR
// ------ KNXnet/IP header
stResult.aMessage[1] 	:= E_KNXnetIP_COMMON_CONSTANTS.HEADER_SIZE_10;
stResult.aMessage[2] 	:= E_KNXnetIP_COMMON_CONSTANTS.KNXNETIP_VERSION_10;
stResult.aMessage[3] 	:= M_GetHighByte(E_KNXnetIP_TUNNELING.TUNNELING_ACK);
stResult.aMessage[4] 	:= M_GetLowByte(E_KNXnetIP_TUNNELING.TUNNELING_ACK);
stResult.aMessage[5] 	:= M_GetHighByte(cTotalLength);
stResult.aMessage[6] 	:= M_GetLowByte(cTotalLength);
stResult.aMessage[7]	:= cStructLengthCONNECTIONHEADER;
stResult.aMessage[8]	:= nCommunicationChannelID;
stResult.aMessage[9]	:= P_SequenceCounterReceive;
stResult.aMessage[10]	:= E_KNXnetIP_TUNNELING_CONNECT_ERROR.E_NO_ERROR;

// set length
stResult.nByteLength := WORD_TO_UINT(cTotalLength);

// return result
M_BuildTunnellingAck := stResult;
END_METHOD

METHOD PRIVATE M_BuildTunnellingRequest : ST_KNXnetIP_Message
VAR_INPUT
	stInGroupAddress	: ST_KNX_GroupAddress;		// destination group address
	stInMessage			: ST_KNXnetIP_Message;		// message to send over tunnelling request	
END_VAR
VAR
	stResult			: ST_KNXnetIP_Message;
	nTotalLength		: UINT;
	nByte				: BYTE;
	nWord				: WORD;
	i					: BYTE;
END_VAR
VAR CONSTANT
	cStructLengthCONNECTIONHEADER	: BYTE := 16#04;			// structure length of Connection header are 4 octetts
END_VAR
// ------ KNXnet/IP header
stResult.aMessage[1] 	:= E_KNXnetIP_COMMON_CONSTANTS.HEADER_SIZE_10;
stResult.aMessage[2] 	:= E_KNXnetIP_COMMON_CONSTANTS.KNXNETIP_VERSION_10;
stResult.aMessage[3] 	:= M_GetHighByte(E_KNXnetIP_TUNNELING.TUNNELING_REQUEST);
stResult.aMessage[4] 	:= M_GetLowByte(E_KNXnetIP_TUNNELING.TUNNELING_REQUEST);
nTotalLength := E_KNXnetIP_COMMON_CONSTANTS.HEADER_SIZE_10 + cStructLengthCONNECTIONHEADER + 11 + UDINT_TO_BYTE(stInMessage.nByteLength);

// ------ Connection header
stResult.aMessage[7]		:= cStructLengthCONNECTIONHEADER;
stResult.aMessage[8]		:= nCommunicationChannelID;
stResult.aMessage[9]		:= P_SequenceCounterTransmit;
P_SequenceCounterTransmit	:= P_SequenceCounterTransmit + 1;
stResult.aMessage[10]		:= 16#00;						// reserved

// ------ cEMI frame
stResult.aMessage[11]	:= E_KNXnetIP_ServiceTypes.eL_DataReq;
	// Additional Information Length (AddIL)
stResult.aMessage[12]	:= 16#00;
	// Ctrl1
nByte := 16#BC;// 16#8C;		// 1... .... Frame Type: Standard (1), ..1. .... Repeat On Error: No (1), ...1 .... Broadcast Type: Domain (1), .... 11.. Priority: Low (3), ..... ..0. Ack Wanted: No (0), .... ...0 Confirmation Error: No (0)
stResult.aMessage[13]	:= nByte;
	// Ctrl2
nByte := 16#E0; // 16#80;		// 1... .... Address Type: Group (1), .000 .... Hop Count: 0, .... 0000 Extended Frame Format: 0x0
stResult.aMessage[14]	:= nByte;
	// Source
nWord := F_KNX_PHYSICALADDRESS_TO_WORD(stInPhysicalAddress);
stResult.aMessage[15]	:= M_GetHighByte(nWord);	// 0x00 means that the server will send his own source physical address
stResult.aMessage[16]	:= M_GetLowByte(nWord);		// 0x00 means that the server will send his own source physical address
	// Destination
nWord := F_KNX_GROUPADDRESS_TO_WORD(stInGroupAddress);
stResult.aMessage[17]	:= M_GetHighByte(nWord);
stResult.aMessage[18]	:= M_GetLowByte(nWord);
	// Length, number of NPDU octets, TPCI octet not included!
stResult.aMessage[19]	:= UDINT_TO_BYTE(stInMessage.nByteLength+1);
	// TPCI/APCI
stResult.aMessage[20]	:= 16#00;
stResult.aMessage[21]	:= 16#80;	// GroupValueWrite
IF stInMessage.nByteLength = 0 THEN
	stResult.aMessage[21]	:= stResult.aMessage[21] OR stInMessage.aMessage[1];
ELSE
	FOR i := 1 TO UDINT_TO_BYTE(stInMessage.nByteLength) DO
		stResult.aMessage[21 + i] := stInMessage.aMessage[i];
	END_FOR
END_IF



// set length
stResult.aMessage[5] 	:= M_GetHighByte(nTotalLength);
stResult.aMessage[6] 	:= M_GetLowByte(nTotalLength);
stResult.nByteLength := WORD_TO_UINT(nTotalLength);

// return result
M_BuildTunnellingRequest := stResult;
END_METHOD

METHOD M_Connect : BOOL
VAR
	bResult 		: BOOL;
END_VAR
IF P_G_IsConnected THEN
	bResult := TRUE;
ELSIF P_G_IsConnecting THEN
	;
ELSIF NOT P_G_IsConnected AND NOT P_G_IsDisconnecting THEN
	bInitiateConnection		:= TRUE;
END_IF

M_Connect := bResult;
END_METHOD

METHOD M_Disconnect : BOOL
VAR
	bResult 		: BOOL;
END_VAR
IF NOT P_G_IsConnected THEN
	bResult := TRUE;
ELSIF P_G_IsDisconnecting THEN
	;
ELSIF P_G_IsConnected AND NOT P_G_IsConnecting THEN
	bInitiateDisconnection		:= TRUE;
END_IF

M_Disconnect := bResult;
END_METHOD

METHOD PRIVATE M_GetHeader : BOOL
VAR_INPUT
END_VAR
END_METHOD

METHOD PRIVATE M_GetHighByte : BYTE
VAR_INPUT
	nWord		: WORD;
END_VAR
VAR
	nResult		: BYTE;
END_VAR
nResult 		:= WORD_TO_BYTE(SHR(nWord, 8));
M_GetHighByte 	:= nResult;
END_METHOD

METHOD PRIVATE M_GetLowByte : BYTE
VAR_INPUT
	nWord		: WORD;
END_VAR
VAR
	nResult		: BYTE;
END_VAR
nResult 		:= WORD_TO_BYTE(nWord AND 16#FF);
M_GetLowByte 	:= nResult;
END_METHOD

METHOD PRIVATE M_Init : BOOL
VAR_INPUT
END_VAR
// reset buffer
fbReceiveFiFoBuffer.M_Reset();

bInit := FALSE;
END_METHOD

METHOD PRIVATE M_IsCEMI_L_DataCon : BOOL
VAR_INPUT
	stInMessage		: ST_KNXnetIP_Message;
END_VAR
VAR
	bResult			: BOOL;
END_VAR
IF stInMessage.aMessage[11] = E_KNXnetIP_ServiceTypes.eL_DataCon THEN
	bResult := TRUE;
END_IF
M_IsCEMI_L_DataCon := bResult;
END_METHOD

METHOD PRIVATE M_IsCEMI_L_DataInd : BOOL
VAR_INPUT
	stInMessage		: ST_KNXnetIP_Message;
END_VAR
VAR
	bResult			: BOOL;
END_VAR
IF stInMessage.aMessage[11] = E_KNXnetIP_ServiceTypes.eL_DataInd THEN
	bResult := TRUE;
END_IF
M_IsCEMI_L_DataInd := bResult;
END_METHOD

METHOD PRIVATE M_IsConnectionStateResponseValid : BOOL
VAR_INPUT
	stInMessage		: ST_KNXnetIP_Message;
END_VAR
VAR_OUTPUT
	nErrorCode		: E_KNXnetIP_CONNECTIONSTATE_RESPONSE_ERROR;
END_VAR
VAR
	bResult			: BOOL;
	stResponse		: ST_KNXnetIP_ConnectionStateResponse;
END_VAR
IF M_ParseServiceType(stInMessage) = E_KNXnetIP_CORE.CONNECTIONSTATE_RESPONSE THEN
	stResponse := M_ParseConnectionStateResponse(stInMessage);
	
	nErrorCode := stResponse.nStatusCode;
	IF stResponse.nStatusCode = E_KNXnetIP_CONNECTIONSTATE_RESPONSE_ERROR.E_NO_ERROR THEN
		bResult := TRUE;
	ELSE
		; 	// errors
	END_IF
END_IF
M_IsConnectionStateResponseValid := bResult;
END_METHOD

METHOD PRIVATE M_IsConnectResponseValid : BOOL
VAR_INPUT
	stInMessage		: ST_KNXnetIP_Message;
END_VAR
VAR
	bResult			: BOOL;
	stResponse		: ST_KNXnetIP_ConnectResponse;
END_VAR
IF M_ParseServiceType(stInMessage) = E_KNXnetIP_CORE.CONNECT_RESPONSE THEN
	stResponse := M_ParseConnectResponse(stInMessage);
	
	IF stResponse.nStatusCode = E_KNXnetIP_CONNECT_RESPONSE_ERROR.E_NO_ERROR THEN
		// store necessary data
		nCommunicationChannelID 	:= stResponse.nCommunicationChannelID;
		M_SetPhysicalAddressTunnelingServer(stResponse.nPhysicalAddress);

		bResult := TRUE;
	ELSE
		; 	// errors
	END_IF
END_IF

M_IsConnectResponseValid := bResult;
END_METHOD

METHOD PRIVATE M_IsDisconnectReqValid : BOOL
VAR_INPUT
	stInMessage		: ST_KNXnetIP_Message;
END_VAR
VAR
	bResult			: BOOL;
	stRequest		: ST_KNXnetIP_DisconnectRequest;
	aIPv4Address	: T_IPv4AddrArr;			// ipv4 address in bytes
	nDWord			: DWORD;
END_VAR
IF M_ParseServiceType(stInMessage) = E_KNXnetIP_CORE.DISCONNECT_REQUEST THEN
	// check the correct channel id, also
	stRequest 		:= M_ParseDisconnectRequest(stInMessage);
	aIPv4Address	:= F_ScanIPv4AddrIds(sInRemoteHostIPv4Addr);
	nDWord	:= SHL(TO_DWORD(aIPv4Address[0]), 8*3);
	nDWord	:= nDWord OR SHL(TO_DWORD(aIPv4Address[1]), 8*2);
	nDWord	:= nDWord OR SHL(TO_DWORD(aIPv4Address[2]), 8);
	nDWord	:= nDWord OR TO_DWORD(aIPv4Address[3]);
	
	IF stRequest.nControlEndpointIPv4 = nDWord AND nCommunicationChannelID = stRequest.nCommunicationChannelID THEN
		bResult := TRUE;
	END_IF
END_IF

M_IsDisconnectReqValid := bResult;
END_METHOD

METHOD PRIVATE M_IsDisconnectResponseValid : BOOL
VAR_INPUT
	stInMessage		: ST_KNXnetIP_Message;
END_VAR
VAR
	bResult			: BOOL;
	stResponse		: ST_KNXnetIP_DisconnectResponse;
END_VAR
IF M_ParseServiceType(stInMessage) = E_KNXnetIP_CORE.DISCONNECT_RESPONSE THEN
	stResponse := M_ParseDisconnectResponse(stInMessage);
	
// 	IF stResponse.nStatusCode = E_KNXnetIP_CONNECT_RESPONSE_ERROR.E_NO_ERROR THEN
		// clear storee necessary data
		nCommunicationChannelID 	:= 16#0;
		M_SetPhysicalAddressTunnelingServer(16#0);

		bResult := TRUE;
// 	ELSE
// 		; 	// errors
// 	END_IF
END_IF

M_IsDisconnectResponseValid := bResult;
END_METHOD

METHOD PRIVATE M_IsTunnellingAckValid: BOOL
VAR_INPUT
	stInMessage		: ST_KNXnetIP_Message;
END_VAR
VAR
	bResult				: BOOL;
END_VAR
IF M_ParseServiceType(stInMessage) = E_KNXnetIP_TUNNELING.TUNNELING_ACK THEN
	bResult := TRUE;
END_IF

M_IsTunnellingAckValid := bResult;
END_METHOD

METHOD PRIVATE M_IsTunnellingReqValid : BOOL
VAR_INPUT
	stInMessage		: ST_KNXnetIP_Message;
END_VAR
VAR
	bResult				: BOOL;
	nStartByteConHeader	: UINT := 7;
END_VAR
IF M_ParseServiceType(stInMessage) = E_KNXnetIP_TUNNELING.TUNNELING_REQUEST THEN
	M_RefreshSequenceCounter(M_ParseConnectionHeader(stInMessage, nStartByteConHeader));
	bResult := TRUE;
END_IF

M_IsTunnellingReqValid := bResult;
END_METHOD

METHOD PRIVATE M_ManagerConnection : BOOL
VAR_INST
	eState							: E_KNXnetIPStateConnection;			// state machine for connection to tunneling server
	                                                                		
	bInit							: BOOL := TRUE;                 		
	                                                                		
	// udp connection                                               		
	fbCloseSocket					: FB_SocketClose;						// will close the open TCP/UDP/IP socket
	fbCloseAllSockets				: FB_SocketCloseAll;					// will close all TCP/UDP/IP sockets
	fbCreateUdpSocket				: FB_SocketUdpCreate;					// create a new udp socket for communication
	tnWaitForResponse				: TON;									// timer to wait for connect response
	tnNextConnectionStateRequest	: TON;									// timer to send next connection state request, to keep connection alive
	stMessage						: ST_KNXnetIP_Message;					// message for KNXnetIP
	nCountFailedConStateResponses	: UINT;									// counter for failed connection state responses
	nErrorCounter					: UINT;									// error counter 
END_VAR
VAR CONSTANT
	ctTimeout						: TIME := T#5S;
	stSocketClear					: T_HSOCKET;
	ctTimeoutNextConnectionRequest	: TIME := CONNECTION_HEARTBEAT_TIME;	// time to send next connection request, to kepp connection alive
	cnMaxFailedConStateResponses	: UINT := 3;							// max count of failed connection responses
END_VAR
IF bInit THEN
	fbCloseSocket( bExecute := FALSE);
	bInit := FALSE;
END_IF

// disconnecting request received
IF P_DisconnectReceived THEN
	P_DisconnectReceived := FALSE;
	eState := E_KNXnetIPStateConnection.eAckDisconnectReq;
END_IF

CASE eState OF
	
// init, with deletion of existing socket handle -------------------------------------------------------------------------------------------------
	E_KNXnetIPStateConnection.eInit:
		M_Reset();
		nCountFailedConStateResponses	:= 0;
		nErrorCounter					:= 0;
		P_SequenceCounterTransmit		:= 0;
		fbTransmitFiFoBuffer.M_Reset();
		fbTransmitFiFoBufferQuick.M_Reset();
	
			// close open socket if needed
		IF P_Socket.handle <> 0 AND NOT fbCloseSocket.bError THEN			
			fbCloseSocket( sSrvNetId	:= sInSrvNetId,
							hSocket		:= P_Socket,
							bExecute	:= TRUE,
							tTimeout	:= ctTimeout);
		END_IF
		
			// clear connected socket
		IF NOT fbCloseSocket.bBusy AND NOT fbCloseSocket.bError THEN
			_stConnectedSocket := stSocketClear;
			fbCloseSocket(bExecute := FALSE);
		END_IF
			// repeat if error occur
		IF fbCloseSocket.bError THEN
			fbCloseSocket(bExecute := FALSE);
			IF fbCloseSocket.nErrId = 16#8002 THEN
				_stConnectedSocket := stSocketClear;
			END_IF
		END_IF
		
			// initiate new udp connection
		IF bInitiateConnection AND P_Socket.handle = 0 THEN
			bInitiateConnection	:= FALSE;			
			fbCreateUdpSocket(bExecute := FALSE);
			P_G_IsConnecting	:= TRUE;
			eState 	:= E_KNXnetIPStateConnection.eCreateUdpSocket;
		END_IF
		
// create udp socket for connection-------------------------------------------------------------------------------------------------
	E_KNXnetIPStateConnection.eCreateUdpSocket:
		fbCreateUdpSocket(	sSrvNetId		:= sInSrvNetId,
							sLocalHost		:= sInLocalHostIPv4Addr,
							nLocalPort		:= nInLocalPort,
							bExecute		:= TRUE,
							tTimeout		:= ctTimeout);
			// wait udp socket is created
		IF NOT fbCreateUdpSocket.bBusy AND NOT fbCreateUdpSocket.bError THEN
			_stConnectedSocket	:= fbCreateUdpSocket.hSocket;
			fbCreateUdpSocket(bExecute := FALSE);
			eState 		:= E_KNXnetIPStateConnection.eSendConnectRequestToTunnelingServer;
		END_IF
			// if error occur, repeat delete socket and try again
		IF fbCreateUdpSocket.bError THEN			
			bInitiateConnection	:= TRUE;
			fbCreateUdpSocket(bExecute := FALSE);
			
				// error this socket is already in use
			IF fbCreateUdpSocket.nErrId = 16#80072740 THEN
				fbCloseAllSockets(bExecute := FALSE);
				eState	:= E_KNXnetIPStateConnection.eCloseAllSockets;
			ELSE				
				eState	:= E_KNXnetIPStateConnection.eInit;
			END_IF	
		
		END_IF
		
// send request to connecting to tunneling server -------------------------------------------------------------------------------------------------
	E_KNXnetIPStateConnection.eSendConnectRequestToTunnelingServer:
		
		fbTransmitFiFoBufferQuick.M_Append(M_BuildTunnelConnectRequest());
		tnWaitForResponse(IN := FALSE);
		eState := E_KNXnetIPStateConnection.eWaitForConnectResponse;
		
// wait for response of tunneling server -------------------------------------------------------------------------------------------------
	E_KNXnetIPStateConnection.eWaitForConnectResponse:
		
		IF P_ConnectResponseReceived THEN
			P_ConnectResponseReceived := FALSE;
				// connection response was valid
			eState := E_KNXnetIPStateConnection.eConnected;
			P_G_IsConnecting 	:= FALSE;
			P_G_IsConnected 	:= TRUE;
		END_IF
	
		tnWaitForResponse(IN := TRUE, PT := CONNECT_REQUEST_TIMEOUT);
			// too long time for response
		IF tnWaitForResponse.Q THEN
			tnWaitForResponse(IN := FALSE);
				// repeat tunneling connection request
			eState := E_KNXnetIPStateConnection.eSendConnectRequestToTunnelingServer;
		END_IF
	
// connected, than wait for sending next connection  -------------------------------------------------------------------------------------------------	
	E_KNXnetIPStateConnection.eConnected:
		tnNextConnectionStateRequest(IN := TRUE, PT := ctTimeoutNextConnectionRequest);
		
		IF tnNextConnectionStateRequest.Q THEN
			tnNextConnectionStateRequest(IN := FALSE);
			eState := E_KNXnetIPStateConnection.eSendConnectionStateRequest;
		END_IF
		
			// disconnecting valid connection
		IF bInitiateDisconnection THEN
			tnNextConnectionStateRequest(IN := FALSE);
			bInitiateDisconnection 	:= FALSE;
			P_G_IsDisconnecting		:= TRUE;
			eState := E_KNXnetIPStateConnection.eDisconnectValidConnection;
		ELSIF P_Reconnect THEN
			tnNextConnectionStateRequest(IN := FALSE);
			P_Reconnect := FALSE;	
				// delete connection and initiate new connection
			bInitiateConnection := TRUE;
			eState := E_KNXnetIPStateConnection.eDisconnectValidConnection;
		END_IF
		
// send connection state request to server -------------------------------------------------------------------------------------------------	
	E_KNXnetIPStateConnection.eSendConnectionStateRequest:	
		
		fbTransmitFiFoBufferQuick.M_Append(M_BuildTunnelConnectionStateRequest());
		tnWaitForResponse(IN := FALSE);
		eState 			:= E_KNXnetIPStateConnection.eWaitForConnectionStateResponse;
		
// wait for connection state response from server -------------------------------------------------------------------------------------------------	
	E_KNXnetIPStateConnection.eWaitForConnectionStateResponse:	
	
		IF P_ConnectionStateResponseReceived THEN
			P_ConnectionStateResponseReceived 	:= FALSE;
			nCountFailedConStateResponses		:= 0;
			tnWaitForResponse(IN := FALSE);
				// connection state response was valid
			eState := E_KNXnetIPStateConnection.eConnected;
		END_IF
	
		tnWaitForResponse(IN := TRUE, PT := CONNECTIONSTATE_REQUEST_TIMEOUT);
			// too long time for response
		IF tnWaitForResponse.Q THEN
			tnWaitForResponse(IN := FALSE);
			IF nCountFailedConStateResponses > cnMaxFailedConStateResponses THEN
					// delete connection and initiate new connection
				bInitiateConnection := TRUE;
				eState := E_KNXnetIPStateConnection.eInit;
			ELSE
					// try new request again
				nCountFailedConStateResponses := nCountFailedConStateResponses + 1;
				eState := E_KNXnetIPStateConnection.eSendConnectionStateRequest;				
			END_IF
		ELSIF P_Reconnect THEN
			P_Reconnect := FALSE;	
				// delete connection and initiate new connection
			bInitiateConnection := TRUE;
			eState := E_KNXnetIPStateConnection.eDisconnectValidConnection;
		END_IF

// disconnect valid connection -------------------------------------------------------------------------------------------------	
	E_KNXnetIPStateConnection.eDisconnectValidConnection:
	
		fbTransmitFiFoBufferQuick.M_Append(M_BuildTunnelDisconnectRequest());
		tnWaitForResponse(IN := FALSE);
		eState := E_KNXnetIPStateConnection.eWaitForDisconnectResponse;
		
// wait for disconnect response from server -------------------------------------------------------------------------------------------------	
	E_KNXnetIPStateConnection.eWaitForDisconnectResponse:	

		IF P_DisconnectResponseReceived THEN
			P_DisconnectResponseReceived := FALSE;
				// connection state response was valid
			eState := E_KNXnetIPStateConnection.eInit;
		END_IF
	
		tnWaitForResponse(IN := TRUE, PT := T#1S);
			// too long time for response
		IF tnWaitForResponse.Q THEN
			tnWaitForResponse(IN := FALSE);
				// delete connection and initiate new connection
			eState := E_KNXnetIPStateConnection.eInit;
		END_IF
		
// ack disconnect request -------------------------------------------------------------------------------------------------	
	E_KNXnetIPStateConnection.eAckDisconnectReq:
			// clear storee necessary data
		nCommunicationChannelID 	:= 16#0;
		M_SetPhysicalAddressTunnelingServer(16#0);
		bInitiateConnection			:= TRUE;		// try new connecting
		eState := E_KNXnetIPStateConnection.eInit;

	
// close all sockets if needed -------------------------------------------------------------------------------------------------	
	E_KNXnetIPStateConnection.eCloseAllSockets:		
		
		fbCloseAllSockets(bExecute := TRUE);
		IF NOT fbCloseAllSockets.bBusy THEN
			fbCloseAllSockets(bExecute := FALSE);
			eState := E_KNXnetIPStateConnection.eInit;
		END_IF
	
// error
	E_KNXnetIPStateConnection.eError:
		
		;
		
ELSE
	;
END_CASE
END_METHOD

METHOD PRIVATE M_ManagerConvertReceived : BOOL
VAR_INST
	stMessage			: ST_KNXnetIP_Message;
	stcEMI_L_DataInd	: ST_KNXnetIP_cEMI;
	stcEMI_L_DataCon	: ST_KNXnetIP_cEMI;
END_VAR
MEMSET(ADR(stGroupAddressMessages.aNewMessage), 0, SIZEOF(stGroupAddressMessages.aNewMessage));

IF fbReceiveFiFoBuffer.P_G_Count > 0 THEN
	IF M_IsTunnellingReqValid(fbReceiveFiFoBuffer.M_Look()) THEN
		stMessage := fbReceiveFiFoBuffer.M_Drop();
		IF M_IsCEMI_L_DataInd(stMessage) THEN
			stcEMI_L_DataInd := M_ParseTunnellingRequest(stMessage);
			stGroupAddressMessages.aMessage[stcEMI_L_DataInd.stDestinationGroupAddress.nFirst,
												stcEMI_L_DataInd.stDestinationGroupAddress.nMiddle,
												stcEMI_L_DataInd.stDestinationGroupAddress.nLow] := stcEMI_L_DataInd.Data;
			stGroupAddressMessages.aNewMessage[stcEMI_L_DataInd.stDestinationGroupAddress.nFirst,
												stcEMI_L_DataInd.stDestinationGroupAddress.nMiddle,
												stcEMI_L_DataInd.stDestinationGroupAddress.nLow] := TRUE;
			stGroupAddressMessages.aTimeStamp[stcEMI_L_DataInd.stDestinationGroupAddress.nFirst,
												stcEMI_L_DataInd.stDestinationGroupAddress.nMiddle,
												stcEMI_L_DataInd.stDestinationGroupAddress.nLow] := DateAndTime;
		END_IF
	
	ELSIF M_IsTunnellingReqValid(fbReceiveFiFoBuffer.M_LookLast()) THEN
		stMessage := fbReceiveFiFoBuffer.M_DropLast();
		IF M_IsCEMI_L_DataInd(stMessage) THEN
			stcEMI_L_DataInd := M_ParseTunnellingRequest(stMessage);
			stGroupAddressMessages.aMessage[stcEMI_L_DataInd.stDestinationGroupAddress.nFirst,
												stcEMI_L_DataInd.stDestinationGroupAddress.nMiddle,
												stcEMI_L_DataInd.stDestinationGroupAddress.nLow] := stcEMI_L_DataInd.Data;
			stGroupAddressMessages.aNewMessage[stcEMI_L_DataInd.stDestinationGroupAddress.nFirst,
												stcEMI_L_DataInd.stDestinationGroupAddress.nMiddle,
												stcEMI_L_DataInd.stDestinationGroupAddress.nLow] := TRUE;
			stGroupAddressMessages.aTimeStamp[stcEMI_L_DataInd.stDestinationGroupAddress.nFirst,
												stcEMI_L_DataInd.stDestinationGroupAddress.nMiddle,
												stcEMI_L_DataInd.stDestinationGroupAddress.nLow] := DateAndTime;
		ELSIF M_IsCEMI_L_DataCon(stMessage) THEN
			stcEMI_L_DataCon := M_ParseTunnellingRequest(stMessage);
			// confirm bit detection
			IF (stcEMI_L_DataCon.nControlField1 AND 16#01) = 1 THEN
				P_TransmitTimeout := TRUE;
			END_IF
		END_IF
		
	END_IF	


END_IF
END_METHOD

METHOD PRIVATE M_ManagerReceiving : BOOL
VAR_INST
	eState							: E_KNXnetIPStateReceivedTelegrams;	// state machine for receiving telegrams

	// udp receiving
	fbSocketUdpReceive				: FB_SocketUdpReceiveFrom;			// function block for receiving data telegrams over udp
	aBufferReceive					: ST_KNXnetIP_Message;				// receiving buffer
	sRemoteHost						: T_IPv4Addr;						// remote host, which are the data was received
	nRemotePort						: UDINT;							// remote port, which are the data was received
	nErrorCode						: UINT;
END_VAR
CASE eState OF
	
	E_KNXnetIPStateReceivedTelegrams.eInit:
	
		fbSocketUdpReceive(bExecute := FALSE);
		// wait for connection, then it is possible to hear on port for new incomming telegrams
		IF P_G_IsConnecting OR P_G_IsConnected THEN
			eState := E_KNXnetIPStateReceivedTelegrams.eWaitForNextTelegram;
		END_IF
		
	E_KNXnetIPStateReceivedTelegrams.eWaitForNextTelegram:
	
		fbSocketUdpReceive(	sSrvNetId		:= sInSrvNetId,
							hSocket			:= P_Socket,
							cbLen			:= SIZEOF(aBufferReceive.aMessage),
							pDest			:= ADR(aBufferReceive.aMessage[1]),
							bExecute		:= TRUE,
							sRemoteHost		=> sRemoteHost,
							nRemotePort		=> nRemotePort,
							nRecBytes		=> aBufferReceive.nByteLength);
							
		IF NOT fbSocketUdpReceive.bBusy AND NOT fbSocketUdpReceive.bError THEN
			IF M_AreHostAndPortValid(sRemoteHost, nRemotePort) THEN
				IF M_IsDisconnectReqValid(aBufferReceive) THEN
					P_DisconnectReceived := TRUE;
				ELSIF P_G_IsDisconnecting AND M_IsDisconnectResponseValid(aBufferReceive) THEN
					P_DisconnectResponseReceived := TRUE;
				ELSIF P_G_IsConnected AND M_IsConnectionStateResponseValid(aBufferReceive, nErrorCode => nErrorCode) OR_ELSE nErrorCode <> E_KNXnetIP_CONNECTIONSTATE_RESPONSE_ERROR.E_NO_ERROR THEN
					IF nErrorCode <> E_KNXnetIP_CONNECTIONSTATE_RESPONSE_ERROR.E_NO_ERROR THEN
						P_Reconnect := TRUE;
					ELSE						
						P_ConnectionStateResponseReceived := TRUE;
					END_IF
				ELSIF P_G_IsConnecting AND M_IsConnectResponseValid(aBufferReceive) THEN
					P_ConnectResponseReceived := TRUE;
				ELSIF M_IsTunnellingAckValid(aBufferReceive) THEN
					P_TunnellingAckReceived := TRUE;
				ELSIF M_IsTunnellingReqValid(aBufferReceive) THEN
					P_TunnellingReqReceived := TRUE;
						// if host and port valid, then append the message to local receive buffer. In this case it is not possible to overload the buffer.
					fbReceiveFiFoBuffer.M_Append(aBufferReceive);
				END_IF				
			END_IF
				// next receiving of data
			fbSocketUdpReceive(bExecute := FALSE);
		ELSIF fbSocketUdpReceive.bError THEN
				// try receiving again
			fbSocketUdpReceive(bExecute := FALSE);
		END_IF

ELSE
	;
END_CASE
END_METHOD

METHOD PRIVATE M_ManagerTransmit : BOOL
VAR_INST
	eState							: E_KNXnetIPStateTransmitTelegrams;	// state machine for transmitting telegrams

	//	// udp connection
	fbSendToUdpSocket				: FB_SocketUdpSendTo;				// function block to send messages to the connected udp socket
	stMessage						: ST_KNXnetIP_Message;				// message for KNXnetIP

	stStoredTunnellingReq			: ST_KNXnetIP_Message;				// stored message to send this to server again
	bIsWaitingForTunnellingAck		: BOOL;								// next tunneling telegram only send if Ack from first is received
	tnWaitTunnellingAck				: TON;								// timer for waiting of tunnelling ack from server
	nCountWaitTunnellingAck			: UINT;								// counter for waiting of tunnelling ack from server
	aBufferLookLast					: ST_KNXnetIP_Message;				// last message in buffer, if with high priority than send this first
	tnWaitTimeNextTransmit			: TON;								// timer for next transmit
END_VAR
VAR CONSTANT
	stClear							: ST_KNXnetIP_Message;
END_VAR
// reset State to init, if no valid socket available
IF P_Socket.handle = 0 THEN
	eState 						:= E_KNXnetIPStateTransmitTelegrams.eInit;
	stMessage					:= stClear;
	bIsWaitingForTunnellingAck	:= FALSE;
END_IF

// waiting timer for ack from server if tunnelling request was send
tnWaitTunnellingAck(IN := bIsWaitingForTunnellingAck, PT := KNXnetIP_TIMEOUT_CONSTANS.TUNNELING_REQUEST_TIMEOUT);

CASE eState OF
	
	E_KNXnetIPStateTransmitTelegrams.eInit:
	
		fbSendToUdpSocket(bExecute := FALSE);
		// wait for connection, then it is possible to transmit new telegrams
		IF P_G_IsConnecting OR P_G_IsConnected THEN
			eState := E_KNXnetIPStateTransmitTelegrams.eWaitForNextTelegramToTransmit;
		END_IF
		
	E_KNXnetIPStateTransmitTelegrams.eWaitForNextTelegramToTransmit:
	
		fbSendToUdpSocket(bExecute := FALSE);
		
			// disconnect response
		IF P_DisconnectReceived THEN
			P_DisconnectReceived 		:= FALSE;
			stMessage					:= M_BuildDisconnectResponse();
			fbTransmitFiFoBuffer.M_Reset();
			// tunnelling request received
		ELSIF P_TunnellingReqReceived THEN
			P_TunnellingReqReceived		:= FALSE;
			stMessage					:= M_BuildTunnellingAck();
			// tunnelling ack received
		ELSIF P_TunnellingAckReceived THEN
			P_TunnellingAckReceived		:= FALSE;
			bIsWaitingForTunnellingAck	:= FALSE;
			nCountWaitTunnellingAck		:= 0;
		ELSIF tnWaitTunnellingAck.Q THEN
			IF nCountWaitTunnellingAck > 1 THEN
				nCountWaitTunnellingAck 	:= 0;
				bIsWaitingForTunnellingAck	:= FALSE;
				P_Reconnect := TRUE;
			ELSE
				stMessage 					:= stStoredTunnellingReq;			// do not count sequence counter
				nCountWaitTunnellingAck		:= nCountWaitTunnellingAck + 1;
				bIsWaitingForTunnellingAck	:= FALSE;
			END_IF
		ELSE		
			IF fbTransmitFiFoBufferQuick.P_G_Count > 0 THEN
				stMessage	:= fbTransmitFiFoBufferQuick.M_Drop();
			END_IF
			IF NOT P_Reconnect AND fbTransmitFiFoBuffer.P_G_Count > 0 THEN					
				IF NOT M_IsTunnellingReqValid(fbTransmitFiFoBuffer.M_Look()) THEN
					stMessage	:= fbTransmitFiFoBuffer.M_Drop();
				ELSIF M_IsTunnellingReqValid(fbTransmitFiFoBuffer.M_Look()) AND NOT bIsWaitingForTunnellingAck THEN
					stMessage					:= fbTransmitFiFoBuffer.M_Drop();
					stStoredTunnellingReq		:= stMessage;
					nCountWaitTunnellingAck		:= nCountWaitTunnellingAck + 1;			
				END_IF
			END_IF
		END_IF
		
		IF stClear.nByteLength <> stMessage.nByteLength THEN
			eState := E_KNXnetIPStateTransmitTelegrams.eTransmit;
		END_IF
	
	E_KNXnetIPStateTransmitTelegrams.eTransmit:	
	
		fbSendToUdpSocket(	sSrvNetId	:= sInSrvNetId,
							hSocket		:= P_Socket,
							sRemoteHost	:= sInRemoteHostIPv4Addr,
							nRemotePort	:= nInRemotePort,
							cbLen		:= stMessage.nByteLength,
							pSrc		:= ADR(stMessage.aMessage[1]),
							bExecute	:= TRUE);
	
		IF NOT fbSendToUdpSocket.bBusy AND NOT fbSendToUdpSocket.bError THEN		
			tnWaitTimeNextTransmit(IN := FALSE);	
				// if necessary stop transmitting with timeout		
				eState := E_KNXnetIPStateTransmitTelegrams.eWaitForNextTelegramToTransmit;
			IF M_IsTunnellingReqValid(stMessage) THEN
				bIsWaitingForTunnellingAck := TRUE;
			END_IF
			stMessage 	:= stClear;
		ELSIF fbSendToUdpSocket.bError THEN
			stMessage 	:= stClear;
			eState 		:= E_KNXnetIPStateTransmitTelegrams.eWaitTimeForNextTransmit;
		END_IF	

	
	E_KNXnetIPStateTransmitTelegrams.eWaitTimeForNextTransmit:		

		tnWaitTimeNextTransmit(IN := TRUE, PT := T#100MS);
		IF tnWaitTimeNextTransmit.Q THEN		
			tnWaitTimeNextTransmit(IN := FALSE);			
			eState := E_KNXnetIPStateTransmitTelegrams.eWaitForNextTelegramToTransmit;
		END_IF

ELSE
	;
END_CASE
END_METHOD

METHOD PRIVATE M_Parse_cEMI_L_DataCon : ST_KNXnetIP_cEMI
VAR_INPUT
	stInMessage		: ST_KNXnetIP_Message;
	nStartByte		: UINT;
END_VAR
VAR
	i				: UINT;
END_VAR
VAR_INST
	stResult		: ST_KNXnetIP_cEMI;
	nWord			: WORD;
	nFollowOctets	: BYTE;
END_VAR
stResult.nMessageCode				:= stInMessage.aMessage[nStartByte];
stResult.nAdditionalInfoLength		:= stInMessage.aMessage[nStartByte+1];
// IF stResult.nAdditionalInfoLength > 16#0 THEN
// 	stResult.nAdditionalInfo			:= stInMessage.aMessage[nStartByte];
// END_IF
stResult.nControlField1				:= stInMessage.aMessage[nStartByte+2+stResult.nAdditionalInfoLength];
stResult.nControlField2				:= stInMessage.aMessage[nStartByte+3+stResult.nAdditionalInfoLength];
nWord := SHL(BYTE_TO_WORD(stInMessage.aMessage[nStartByte+4+stResult.nAdditionalInfoLength]), 8);
nWord := nWord OR BYTE_TO_WORD(stInMessage.aMessage[nStartByte+5+stResult.nAdditionalInfoLength]);
stResult.nSourcePhysicalAddress 	:= nWord;
stResult.stSourcePhysicalAddress	:= F_WORD_TO_KNX_PHYSICALADDRESS(nWord);


nWord := SHL(BYTE_TO_WORD(stInMessage.aMessage[nStartByte+6+stResult.nAdditionalInfoLength]), 8);
nWord := nWord OR BYTE_TO_WORD(stInMessage.aMessage[nStartByte+7+stResult.nAdditionalInfoLength]);
stResult.nDestinationGroupAddress	:= nWord;
stResult.stDestinationGroupAddress	:= F_WORD_TO_KNX_GROUPADDRESS(nWord);

stResult.LengthDataField			:= stInMessage.aMessage[nStartByte+8+stResult.nAdditionalInfoLength];
// TPCI is next octet nStartByte+9+stResult.nAdditionalInfoLength, TPCI is not included in LengthDataField!
nFollowOctets := stResult.LengthDataField;
// APCI is next octet nStartByte+10+stResult.nAdditionalInfoLength
nFollowOctets := nFollowOctets - 1;
// fill data fields
IF nFollowOctets > 0 THEN
	FOR i := 1 TO nFollowOctets DO
		stResult.Data[i] := stInMessage.aMessage[nStartByte+10+stResult.nAdditionalInfoLength+i];
	END_FOR
ELSE
	stResult.Data[i] := stInMessage.aMessage[nStartByte+10+stResult.nAdditionalInfoLength] AND 16#1;
END_IF

M_Parse_cEMI_L_DataCon := stResult;
END_METHOD

METHOD PRIVATE M_Parse_cEMI_L_DataInd : ST_KNXnetIP_cEMI
VAR_INPUT
	stInMessage		: ST_KNXnetIP_Message;
	nStartByte		: UINT;
END_VAR
VAR
	i				: UINT;
END_VAR
VAR_INST
	stResult		: ST_KNXnetIP_cEMI;
	nWord			: WORD;
	nFollowOctets	: BYTE;
END_VAR
stResult.nMessageCode				:= stInMessage.aMessage[nStartByte];
stResult.nAdditionalInfoLength		:= stInMessage.aMessage[nStartByte+1];
// IF stResult.nAdditionalInfoLength > 16#0 THEN
// 	stResult.nAdditionalInfo			:= stInMessage.aMessage[nStartByte];
// END_IF
stResult.nControlField1				:= stInMessage.aMessage[nStartByte+2+stResult.nAdditionalInfoLength];
stResult.nControlField2				:= stInMessage.aMessage[nStartByte+3+stResult.nAdditionalInfoLength];
nWord := SHL(BYTE_TO_WORD(stInMessage.aMessage[nStartByte+4+stResult.nAdditionalInfoLength]), 8);
nWord := nWord OR BYTE_TO_WORD(stInMessage.aMessage[nStartByte+5+stResult.nAdditionalInfoLength]);
stResult.nSourcePhysicalAddress 	:= nWord;
stResult.stSourcePhysicalAddress	:= F_WORD_TO_KNX_PHYSICALADDRESS(nWord);


nWord := SHL(BYTE_TO_WORD(stInMessage.aMessage[nStartByte+6+stResult.nAdditionalInfoLength]), 8);
nWord := nWord OR BYTE_TO_WORD(stInMessage.aMessage[nStartByte+7+stResult.nAdditionalInfoLength]);
stResult.nDestinationGroupAddress	:= nWord;
stResult.stDestinationGroupAddress	:= F_WORD_TO_KNX_GROUPADDRESS(nWord);

stResult.LengthDataField			:= stInMessage.aMessage[nStartByte+8+stResult.nAdditionalInfoLength];
// TPCI is next octet nStartByte+9+stResult.nAdditionalInfoLength, TPCI is not included in LengthDataField!
nFollowOctets := stResult.LengthDataField;
// APCI is next octet nStartByte+10+stResult.nAdditionalInfoLength
nFollowOctets := nFollowOctets - 1;
// fill data fields
IF nFollowOctets > 0 THEN
	FOR i := 1 TO nFollowOctets DO
		stResult.Data[i] := stInMessage.aMessage[nStartByte+10+stResult.nAdditionalInfoLength+i];
	END_FOR
ELSE
	stResult.Data[1] := stInMessage.aMessage[nStartByte+10+stResult.nAdditionalInfoLength] AND 16#01;
END_IF

M_Parse_cEMI_L_DataInd := stResult;
END_METHOD

METHOD PRIVATE M_ParseCommonHeader : ST_KNXnetIP_CommonHeader
VAR_INPUT
	stInMessage		: ST_KNXnetIP_Message;
END_VAR
VAR
	stHeader		: ST_KNXnetIP_CommonHeader;
END_VAR
stHeader.nHeaderSize		:= stInMessage.aMessage[1];
stHeader.nProtocolVersion	:= stInMessage.aMessage[2];
stHeader.nServiceType		:= SHL(TO_WORD(stInMessage.aMessage[3]), 8);
stHeader.nServiceType		:= stHeader.nServiceType OR TO_WORD(stInMessage.aMessage[4]);
stHeader.nTotalLength		:= SHL(TO_WORD(stInMessage.aMessage[5]), 8);
stHeader.nTotalLength		:= stHeader.nServiceType OR TO_WORD(stInMessage.aMessage[6]);

M_ParseCommonHeader			:= stHeader;
END_METHOD

METHOD PRIVATE M_ParseConnectionHeader : ST_KNXnetIP_ConnectionHeader
VAR_INPUT
	stInMessage		: ST_KNXnetIP_Message;
	nStartByte		: UINT;
END_VAR
VAR
	stConHeader		: ST_KNXnetIP_ConnectionHeader;
END_VAR
stConHeader.nStructureLength		:= stInMessage.aMessage[nStartByte];
stConHeader.nCommunicationChannel	:= stInMessage.aMessage[nStartByte+1];
stConHeader.nSequenceCounter		:= stInMessage.aMessage[nStartByte+2];
stConHeader.nReserved				:= stInMessage.aMessage[nStartByte+3];

M_ParseConnectionHeader				:= stConHeader;
END_METHOD

METHOD PRIVATE M_ParseConnectionStateResponse : ST_KNXnetIP_ConnectionStateResponse
VAR_INPUT
	stInMessage		: ST_KNXnetIP_Message;
END_VAR
VAR
	stCommonHeader	: ST_KNXnetIP_CommonHeader;
	stConResponse	: ST_KNXnetIP_ConnectionStateResponse;
END_VAR
stCommonHeader 	:= M_ParseCommonHeader(stInMessage);
stConResponse.nHeaderSize		:= stCommonHeader.nHeaderSize;
stConResponse.nProtocolVersion	:= stCommonHeader.nProtocolVersion;
stConResponse.nServiceType		:= stCommonHeader.nServiceType;
stConResponse.nTotalLength		:= stCommonHeader.nTotalLength;

stConResponse.nCommunicationChannelID	:= stInMessage.aMessage[7];
stConResponse.nStatusCode				:= stInMessage.aMessage[8];

M_ParseConnectionStateResponse := stConResponse;
END_METHOD

METHOD PRIVATE M_ParseConnectResponse : ST_KNXnetIP_ConnectResponse
VAR_INPUT
	stInMessage		: ST_KNXnetIP_Message;
END_VAR
VAR
	stCommonHeader	: ST_KNXnetIP_CommonHeader;
	stConResponse	: ST_KNXnetIP_ConnectResponse;
END_VAR
stCommonHeader 	:= M_ParseCommonHeader(stInMessage);
stConResponse.nHeaderSize		:= stCommonHeader.nHeaderSize;
stConResponse.nProtocolVersion	:= stCommonHeader.nProtocolVersion;
stConResponse.nServiceType		:= stCommonHeader.nServiceType;
stConResponse.nTotalLength		:= stCommonHeader.nTotalLength;

stConResponse.nCommunicationChannelID	:= stInMessage.aMessage[7];
stConResponse.nStatusCode				:= stInMessage.aMessage[8];
stConResponse.nStructureLength			:= stInMessage.aMessage[9];
stConResponse.nHostProtocolCode			:= stInMessage.aMessage[10];
stConResponse.nDataEndpointIPv4			:= SHL(TO_DWORD(stInMessage.aMessage[11]), 8*3);
stConResponse.nDataEndpointIPv4			:= stConResponse.nDataEndpointIPv4 OR SHL(TO_DWORD(stInMessage.aMessage[12]), 8*2);
stConResponse.nDataEndpointIPv4			:= stConResponse.nDataEndpointIPv4 OR SHL(TO_DWORD(stInMessage.aMessage[13]), 8);
stConResponse.nDataEndpointIPv4			:= stConResponse.nDataEndpointIPv4 OR TO_DWORD(stInMessage.aMessage[14]);
stConResponse.nDataEndpointPort			:= SHL(TO_WORD(stInMessage.aMessage[15]), 8);
stConResponse.nDataEndpointPort			:= stConResponse.nDataEndpointPort OR TO_WORD(stInMessage.aMessage[16]);
stConResponse.nStructueLengthCRD		:= stInMessage.aMessage[17];
stConResponse.nConnectionTypeCode		:= stInMessage.aMessage[18];
stConResponse.nPhysicalAddress			:= SHL(TO_WORD(stInMessage.aMessage[19]), 8);
stConResponse.nPhysicalAddress			:= stConResponse.nPhysicalAddress OR TO_WORD(stInMessage.aMessage[20]);

M_ParseConnectResponse := stConResponse;
END_METHOD

METHOD PRIVATE M_ParseDisconnectRequest : ST_KNXnetIP_DisconnectRequest
VAR_INPUT
	stInMessage		: ST_KNXnetIP_Message;
END_VAR
VAR
	stCommonHeader	: ST_KNXnetIP_CommonHeader;
	stDisconRequest	: ST_KNXnetIP_DisconnectRequest;
END_VAR
stCommonHeader 	:= M_ParseCommonHeader(stInMessage);
stDisconRequest.nHeaderSize			:= stCommonHeader.nHeaderSize;
stDisconRequest.nProtocolVersion	:= stCommonHeader.nProtocolVersion;
stDisconRequest.nServiceType		:= stCommonHeader.nServiceType;
stDisconRequest.nTotalLength		:= stCommonHeader.nTotalLength;

stDisconRequest.nCommunicationChannelID	:= stInMessage.aMessage[7];
//			:= stInMessage.aMessage[8];		reserved
stDisconRequest.nStructLength			:= stInMessage.aMessage[9];
stDisconRequest.nHostProtocolCode		:= stInMessage.aMessage[10];

stDisconRequest.nControlEndpointIPv4	:= SHL(TO_DWORD(stInMessage.aMessage[11]), 8*3);
stDisconRequest.nControlEndpointIPv4	:= stDisconRequest.nControlEndpointIPv4 OR SHL(TO_DWORD(stInMessage.aMessage[12]), 8*2);
stDisconRequest.nControlEndpointIPv4	:= stDisconRequest.nControlEndpointIPv4 OR SHL(TO_DWORD(stInMessage.aMessage[13]), 8);
stDisconRequest.nControlEndpointIPv4	:= stDisconRequest.nControlEndpointIPv4 OR TO_DWORD(stInMessage.aMessage[14]);
stDisconRequest.nControlEndpointPort	:= SHL(TO_WORD(stInMessage.aMessage[15]), 8);
stDisconRequest.nControlEndpointPort	:= stDisconRequest.nControlEndpointPort OR TO_WORD(stInMessage.aMessage[16]);
stDisconRequest.nCommunicationChannelID	:= stInMessage.aMessage[11];
stDisconRequest.nCommunicationChannelID	:= stInMessage.aMessage[12];

M_ParseDisconnectRequest := stDisconRequest;
END_METHOD

METHOD PRIVATE M_ParseDisconnectResponse : ST_KNXnetIP_DisconnectResponse
VAR_INPUT
	stInMessage		: ST_KNXnetIP_Message;
END_VAR
VAR
	stCommonHeader	: ST_KNXnetIP_CommonHeader;
	stConResponse	: ST_KNXnetIP_DisconnectResponse;
END_VAR
stCommonHeader 	:= M_ParseCommonHeader(stInMessage);
stConResponse.nHeaderSize		:= stCommonHeader.nHeaderSize;
stConResponse.nProtocolVersion	:= stCommonHeader.nProtocolVersion;
stConResponse.nServiceType		:= stCommonHeader.nServiceType;
stConResponse.nTotalLength		:= stCommonHeader.nTotalLength;

stConResponse.nCommunicationChannelID	:= stInMessage.aMessage[7];
stConResponse.nStatusCode				:= stInMessage.aMessage[8];

M_ParseDisconnectResponse := stConResponse;
END_METHOD

METHOD PRIVATE M_ParseServiceType : WORD
VAR_INPUT
	stInMessage		: ST_KNXnetIP_Message;
END_VAR
VAR
	nWord			: WORD;
END_VAR
nWord := SHL(TO_WORD(stInMessage.aMessage[3]), 8);
nWord := nWord OR TO_WORD(stInMessage.aMessage[4]);

M_ParseServiceType := nWord;
END_METHOD

METHOD PRIVATE M_ParseTunnellingRequest : ST_KNXnetIP_cEMI
VAR_INPUT
	stInMessage			: ST_KNXnetIP_Message;
END_VAR
VAR
	stCommonHeader		: ST_KNXnetIP_CommonHeader;
	stConnectionHeader	: ST_KNXnetIP_ConnectionHeader;
	stConResponse		: ST_KNXnetIP_cEMI;
END_VAR
// actually only L_Data.ind is provided
stCommonHeader		:= M_ParseCommonHeader(stInMessage);			// only for debugging parsing
stConnectionHeader	:= M_ParseConnectionHeader(stInMessage, 7);		// only for debugging parsing
IF M_IsCEMI_L_DataInd(stInMessage) THEN
	stConResponse		:= M_Parse_cEMI_L_DataInd(stInMessage, 11);
ELSIF M_IsCEMI_L_DataCon(stInMessage) THEN
	stConResponse		:= M_Parse_cEMI_L_DataCon(stInMessage, 11);
END_IF
M_ParseTunnellingRequest := stConResponse;
END_METHOD

METHOD PRIVATE M_RefreshSequenceCounter : BOOL
VAR_INPUT
	stInConHeader		: ST_KNXnetIP_ConnectionHeader;
END_VAR
// refresh sequence counter with actual value
P_SequenceCounterReceive := stInConHeader.nSequenceCounter;	// connection header sequence counter
END_METHOD

METHOD PRIVATE M_Reset : BOOL
VAR_INPUT
END_VAR
P_ConnectionStateResponseReceived 	:= FALSE;
P_ConnectResponseReceived 			:= FALSE;
P_DisconnectReceived				:= FALSE;
P_DisconnectResponseReceived		:= FALSE;
P_Reconnect							:= FALSE;
P_TunnellingAckReceived				:= FALSE;
P_TunnellingReqReceived				:= FALSE;
P_G_IsConnected 					:= FALSE;
P_G_IsConnecting 					:= FALSE;
P_G_IsDisconnecting					:= FALSE;
P_TransmitTimeout					:= FALSE;
END_METHOD

METHOD PRIVATE M_SetPhysicalAddressTunnelingServer : BOOL
VAR_INPUT
	nInPhysicalAddress		: WORD;			// physical address in word format to convert to local structure
END_VAR
nPhysicalAddressTunneling			:= nInPhysicalAddress;
_stPhysicalAddressTunneling			:= F_WORD_TO_KNX_PHYSICALADDRESS(nInPhysicalAddress);
END_METHOD

// transmitting group address message to tunnelling server
METHOD M_TransmitMessage : BOOL
VAR_INPUT
	stInGroupAddress		: ST_KNX_GroupAddress;			// group address
	stInMessage				: ST_KNXnetIP_Message;			// message to send
END_VAR
VAR
	bSameMessageAsLast		: BOOL;
	i						: UDINT;
	bNewMessage				: BOOL;
END_VAR
VAR_INST
	stLastGroupAddress		: ST_KNX_GroupAddress;			// last stored group address
	stLastMessage			: ST_KNXnetIP_Message;			// last stored knx message
	stMessage				: ST_KNXnetIP_Message;
END_VAR
IF NOT P_G_IsConnected THEN RETURN; END_IF
// only appending possible if connection is done
FOR i := 1 TO SIZEOF(stInMessage.aMessage) DO
	IF stInMessage.aMessage[i] <> P_G_GroupAddressMessages.aMessage[stInGroupAddress.nFirst,stInGroupAddress.nMiddle,stInGroupAddress.nLow][i] THEN
		bNewMessage := TRUE;
		EXIT;
	END_IF
END_FOR
IF bNewMessage THEN
	stMessage := M_BuildTunnellingRequest(stInGroupAddress, stInMessage);
	P_G_GroupAddressMessages.aMessage[stInGroupAddress.nFirst,stInGroupAddress.nMiddle,stInGroupAddress.nLow]:=stInMessage.aMessage;
	fbTransmitFiFoBuffer.M_Append(stMessage);
	stLastGroupAddress 	:= stInGroupAddress;
	stLastMessage		:= stInMessage;
	M_TransmitMessage 	:= TRUE;
END_IF
END_METHOD

{attribute 'monitoring' := 'variable'}
PROPERTY PRIVATE P_ConnectionStateResponseReceived : BOOL
GET
P_ConnectionStateResponseReceived := _bConnectionStateResponseReceived;
END_GET
SET
_bConnectionStateResponseReceived := P_ConnectionStateResponseReceived;
END_SET
END_PROPERTY

{attribute 'monitoring' := 'variable'}
PROPERTY PRIVATE P_ConnectResponseReceived : BOOL
GET
P_ConnectResponseReceived := _bConnectResponseReceived;
END_GET
SET
_bConnectResponseReceived := P_ConnectResponseReceived;
END_SET
END_PROPERTY

{attribute 'monitoring' := 'variable'}
PROPERTY PRIVATE P_DisconnectReceived : BOOL
GET
_bDisconnectReceived := P_DisconnectReceived;
END_GET
SET
P_DisconnectReceived := _bDisconnectReceived;
END_SET
END_PROPERTY

{attribute 'monitoring' := 'variable'}
PROPERTY PRIVATE P_DisconnectResponseReceived : BOOL
GET
P_DisconnectResponseReceived := _bDisconnectResponseReceived;
END_GET
SET
_bDisconnectResponseReceived := P_DisconnectResponseReceived;
END_SET
END_PROPERTY

{attribute 'monitoring' := 'variable'}
PROPERTY P_G_GroupAddressMessages : REFERENCE TO ST_KNXnetIP_MessageOfAllGroupAddresses
GET
P_G_GroupAddressMessages REF= stGroupAddressMessages;
END_GET
END_PROPERTY

{attribute 'monitoring' := 'variable'}
PROPERTY P_G_IsConnected : BOOL
GET
P_G_IsConnected := _bIsConnected;
END_GET
SET // PRIVATE
_bIsConnected := P_G_IsConnected;
END_SET
END_PROPERTY

{attribute 'monitoring' := 'variable'}
PROPERTY P_G_IsConnecting : BOOL
GET
P_G_IsConnecting := _bIsConnecting;
END_GET
SET // PRIVATE
_bIsConnecting := P_G_IsConnecting;
END_SET
END_PROPERTY

{attribute 'monitoring' := 'variable'}
PROPERTY P_G_IsDisconnecting : BOOL
GET
P_G_IsDisconnecting := _bIsDisconnecting;
END_GET
SET // PRIVATE
_bIsDisconnecting := P_G_IsDisconnecting;
END_SET
END_PROPERTY

{attribute 'monitoring' := 'variable'}
PROPERTY P_G_PhysicalAddress : REFERENCE TO ST_KNX_PhysicalAddress
GET
P_G_PhysicalAddress REF= _stPhysicalAddressTunneling;
END_GET
END_PROPERTY

{attribute 'monitoring' := 'variable'}
PROPERTY PRIVATE P_Reconnect : BOOL
GET
P_Reconnect := _bReconnect;
END_GET
SET
_bReconnect := P_Reconnect;
END_SET
END_PROPERTY

{attribute 'monitoring' := 'variable'}
PROPERTY PRIVATE P_SequenceCounterReceive : BYTE
GET
P_SequenceCounterReceive := _nSequenceCounter;
END_GET
SET
_nSequenceCounter := P_SequenceCounterReceive;
END_SET
END_PROPERTY

{attribute 'monitoring' := 'variable'}
PROPERTY PRIVATE P_SequenceCounterTransmit : BYTE
GET
P_SequenceCounterTransmit := _nSequenceCounterTransmit;
END_GET
SET
_nSequenceCounterTransmit := P_SequenceCounterTransmit;
END_SET
END_PROPERTY

{attribute 'monitoring' := 'variable'}
PROPERTY PRIVATE P_Socket : REFERENCE TO T_HSOCKET
GET
P_Socket REF= _stConnectedSocket;
END_GET
END_PROPERTY

{attribute 'monitoring' := 'variable'}
PROPERTY PRIVATE P_TransmitTimeout : BOOL
GET
P_TransmitTimeout := _bTransmitTimeout;
END_GET
SET
_bTransmitTimeout := P_TransmitTimeout;
END_SET
END_PROPERTY

{attribute 'monitoring' := 'variable'}
PROPERTY PRIVATE P_TunnellingAckReceived : BOOL
GET
P_TunnellingAckReceived := _bTunnellingAckReceived;
END_GET
SET
_bTunnellingAckReceived := P_TunnellingAckReceived;
END_SET
END_PROPERTY

{attribute 'monitoring' := 'variable'}
PROPERTY PRIVATE P_TunnellingReqReceived : BOOL
GET
P_TunnellingReqReceived := _bTunnelReqReceived;
END_GET
SET
_bTunnelReqReceived := P_TunnellingReqReceived;
END_SET
END_PROPERTY

END_FUNCTION_BLOCK

// ---- KNXnetIPTunnelingServer/POUs/KNXnetIP_Message_FiFoBuffer.TcPOU
(*
:Description: function block for buffering KNXnetIP_Messages as FiFo
:Instructions for use: only using in KNXnetIPTunnelingServer necessary
*)
FUNCTION_BLOCK KNXnetIP_Message_FiFoBuffer
VAR_INPUT
END_VAR
VAR_OUTPUT
END_VAR
VAR CONSTANT
	cBufferSizeMin		: UINT := 1;
	cBufferSizeMax		: UINT := 100;
END_VAR
VAR
	aBuffer				: ARRAY[cBufferSizeMin..cBufferSizeMax] OF ST_KNXnetIP_Message;
	nPointerLast		: UINT;										// pointer of last added message
	
	// backing
	_nCount				: UINT;
END_VAR

// append new message to buffer
METHOD M_Append : BOOL
VAR_INPUT
	stInMessage		: ST_KNXnetIP_Message;
END_VAR
nPointerLast 	:= nPointerLast + 1;
P_G_Count		:= nPointerLast;
IF nPointerLast > cBufferSizeMax THEN
		// no further appending possible, buffer is full
	M_Append 		:= FALSE;
	nPointerLast 	:= cBufferSizeMax;
	P_G_Count		:= nPointerLast;
	RETURN;
END_IF

	// add new message to buffer
aBuffer[nPointerLast] := stInMessage;
END_METHOD

// return first added message and delete it from buffer
METHOD M_Drop : ST_KNXnetIP_Message
VAR
	stResult		: ST_KNXnetIP_Message;
END_VAR
VAR CONSTANT
	stClear			: ST_KNXnetIP_Message;
END_VAR
stResult 	:= M_Look();
M_Drop 		:= stResult;
IF stResult.nByteLength = stClear.nByteLength THEN 
	RETURN; // no deletion of first message necessary
END_IF		
M_RemoveFirst();
END_METHOD

// return last added message and delete it from buffer
METHOD M_DropLast : ST_KNXnetIP_Message
VAR
	stResult		: ST_KNXnetIP_Message;
END_VAR
VAR CONSTANT
	stClear			: ST_KNXnetIP_Message;
END_VAR
stResult 	:= M_LookLast();
M_DropLast 		:= stResult;
IF stResult.nByteLength = stClear.nByteLength THEN 
	RETURN; // no deletion of last message necessary
END_IF		
M_RemoveLast();
END_METHOD

// return first added message, no deletion of the message from buffer
METHOD M_Look : ST_KNXnetIP_Message
VAR CONSTANT
	stClear			: ST_KNXnetIP_Message;
END_VAR
	// no messages to drop
IF nPointerLast = 0 THEN
	M_Look := stClear;
	RETURN;	
END_IF

M_Look := aBuffer[cBufferSizeMin];		// look first added message of buffer
END_METHOD

// return last added message, no deletion of the message from buffer
METHOD M_LookLast : ST_KNXnetIP_Message
VAR CONSTANT
	stClear			: ST_KNXnetIP_Message;
END_VAR
	// no messages to drop
IF nPointerLast = 0 THEN
	M_LookLast := stClear;
	RETURN;	
END_IF

M_LookLast := aBuffer[nPointerLast];		// look at last buffered message
END_METHOD

METHOD PRIVATE M_RemoveFirst : BOOL
VAR
	i				: UINT;
END_VAR
VAR CONSTANT
	stClear			: ST_KNXnetIP_Message;
END_VAR
	// nothing to remove from buffer
IF nPointerLast <= 0 THEN
	RETURN;
END_IF

IF nPointerLast > 1 THEN
		// move all buffer message one further
	FOR i := cBufferSizeMin TO nPointerLast - 1 DO
		aBuffer[i] := aBuffer[i + 1];
	END_FOR
END_IF
aBuffer[nPointerLast] := stClear;			// clear last buffered message
nPointerLast 	:= nPointerLast - 1;
P_G_Count		:= nPointerLast;
END_METHOD

METHOD PRIVATE M_RemoveLast : BOOL
VAR
	i				: UINT;
END_VAR
VAR CONSTANT
	stClear			: ST_KNXnetIP_Message;
END_VAR
	// nothing to remove from buffer
IF nPointerLast <= 0 THEN
	RETURN;
END_IF
aBuffer[nPointerLast] := stClear;			// clear last buffered message
nPointerLast 	:= nPointerLast - 1;
P_G_Count		:= nPointerLast;
END_METHOD

// reset all buffer data
METHOD M_Reset : BOOL
VAR
	i			: UINT;
END_VAR
VAR CONSTANT
	stClear		: ST_KNXnetIP_Message;
END_VAR
// clear all data in buffer
FOR i := cBufferSizeMin TO cBufferSizeMax DO
	aBuffer[i] := stClear;
END_FOR
nPointerLast 	:= 0;
P_G_Count		:= nPointerLast;

M_Reset := TRUE;
END_METHOD

{attribute 'monitoring' := 'variable'}
PROPERTY P_G_Count : UINT
GET
P_G_Count := _nCount;
END_GET
SET // PRIVATE
_nCount := P_G_Count;
END_SET
END_PROPERTY

END_FUNCTION_BLOCK

// ---- KNXnetIPTunnelingServer/POUs/KNX_DatapointTypes_Builder.TcPOU
(*
:Description: function block for sending regular DPT messages to KNX devices
:Instructions for use: instantiate this function block to use the implemented interface I_KNX_DPT_Builder and its methods to build the KNX messages correctly
*)
FUNCTION_BLOCK KNX_DatapointTypes_Builder IMPLEMENTS I_KNX_DPT_Builder

METHOD M_Build2Bit : ST_KNXnetIP_Message
VAR_INPUT
	bInValueBit1	: BOOL;
	bInValueBit2	: BOOL;
END_VAR
M_Build2Bit.nByteLength := 0 ;//SIZEOF(BYTE);
M_Build2Bit.aMessage[1].0 := bInValueBit1;
M_Build2Bit.aMessage[1].1 := bInValueBit2;
END_METHOD

METHOD M_Build3Byte : ST_KNXnetIP_Message
VAR_INPUT
	nInValue	: DWORD;
END_VAR
M_Build3Byte.nByteLength := SIZEOF(DWORD)-1;
M_Build3Byte.aMessage[1] := DWORD_TO_BYTE(SHR(nInValue,8*3));
M_Build3Byte.aMessage[2] := DWORD_TO_BYTE(SHR(nInValue,8*2));
M_Build3Byte.aMessage[3] := DWORD_TO_BYTE(SHR(nInValue,8*1));
END_METHOD

METHOD M_BuildBool : ST_KNXnetIP_Message
VAR_INPUT
	bInValue	: BOOL;
END_VAR
M_BuildBool.nByteLength := 0;//SIZEOF(BOOL);
M_BuildBool.aMessage[1] := BOOL_TO_BYTE(bInValue);
END_METHOD

METHOD M_BuildDimming : ST_KNXnetIP_Message
VAR_INPUT
	stInValue		: ST_KNX_DPT_ControlDimming;
END_VAR
VAR
	nResult			: BYTE;
END_VAR
M_BuildDimming.nByteLength := SIZEOF(BYTE);
nResult		:= stInValue.nStepCode;
nResult.3 	:= stInValue.bControl;
M_BuildDimming.aMessage[1] := nResult;
END_METHOD

METHOD M_BuildFloat16 : ST_KNXnetIP_Message
VAR_INPUT
	fInValue	: REAL;
END_VAR

VAR
	nValue		: WORD;
	nExponent	: WORD;
	isPositiv	: INT;
END_VAR
M_BuildFloat16.nByteLength := SIZEOF(WORD);
IF fInValue<0 THEN
	isPositiv:=-1;
ELSE
	isPositiv:=1;
END_IF

IF ABS(fInValue) > 20.48 THEN
	nExponent := DINT_TO_WORD(TRUNC((LOG(25*(fInValue*isPositiv))/LOG(2))-9)+1);
ELSE
	nExponent := 0;
END_IF
IF isPositiv<0THEN
	nExponent:=nExponent+16;
END_IF

nValue:=REAL_TO_WORD(ABS(fInValue)/LREAL_TO_REAL(EXPT(2,nExponent))*100) + nExponent*2048;

M_BuildFloat16.aMessage[1] := WORD_TO_BYTE(SHR(nValue,8));
M_BuildFloat16.aMessage[2] := WORD_TO_BYTE(nValue);
END_METHOD

METHOD M_BuildINT16 : ST_KNXnetIP_Message
VAR_INPUT
	nInValue	: INT;
END_VAR
VAR
	nWord		: WORD;
END_VAR
M_BuildINT16.nByteLength := SIZEOF(WORD);
nWord := INT_TO_WORD(nInValue);
M_BuildINT16.aMessage[1] := WORD_TO_BYTE(SHR(nWord,8));
M_BuildINT16.aMessage[2] := WORD_TO_BYTE(nWord);
END_METHOD

METHOD M_BuildINT32 : ST_KNXnetIP_Message
VAR_INPUT
	nInValue	: DINT;
END_VAR
VAR
	nWord		: DWORD;
END_VAR
M_BuildINT32.nByteLength := SIZEOF(DWORD);
nWord := DINT_TO_DWORD(nInValue);
M_BuildINT32.aMessage[1] := DWORD_TO_BYTE(SHR(nWord,8*3));
M_BuildINT32.aMessage[2] := DWORD_TO_BYTE(SHR(nWord,8*2));
M_BuildINT32.aMessage[3] := DWORD_TO_BYTE(SHR(nWord,8));
M_BuildINT32.aMessage[4] := DWORD_TO_BYTE(nWord);
END_METHOD

METHOD M_BuildString : ST_KNXnetIP_Message
VAR_INPUT
	sInValue	: STRING;
END_VAR
VAR
	i 			: INT := 0;
END_VAR
M_BuildString.nByteLength := LIMIT(0,SIZEOF(sInValue),14);

FOR i:=1 TO 15 BY 1 DO
	IF sInValue[i-1] >= 32 AND sInValue[i-1] <= 122 THEN
		M_BuildString.aMessage[i] := sInValue[i-1];
	ELSE
		M_BuildString.aMessage[i] := 0;
	END_IF
END_FOR
END_METHOD

METHOD M_BuildUINT16 : ST_KNXnetIP_Message
VAR_INPUT
	nInValue	: UINT;
END_VAR
VAR
	nWord		: WORD;
END_VAR
M_BuildUINT16.nByteLength := SIZEOF(WORD);
nWord := UINT_TO_WORD(nInValue);
M_BuildUINT16.aMessage[1] := WORD_TO_BYTE(SHR(nWord,8));
M_BuildUINT16.aMessage[2] := WORD_TO_BYTE(nWord);
END_METHOD

METHOD M_BuildUINT32 : ST_KNXnetIP_Message
VAR_INPUT
	nInValue	: UDINT;
END_VAR
VAR
	nWord		: DWORD;
END_VAR
M_BuildUINT32.nByteLength := SIZEOF(DWORD);
nWord := UDINT_TO_DWORD(nInValue);
M_BuildUINT32.aMessage[1] := DWORD_TO_BYTE(SHR(nWord,8*3));
M_BuildUINT32.aMessage[2] := DWORD_TO_BYTE(SHR(nWord,8*2));
M_BuildUINT32.aMessage[3] := DWORD_TO_BYTE(SHR(nWord,8));
M_BuildUINT32.aMessage[4] := DWORD_TO_BYTE(nWord);
END_METHOD

METHOD M_BuildUINT8 : ST_KNXnetIP_Message
VAR_INPUT
	nInValue		: BYTE;
END_VAR
M_BuildUINT8.nByteLength	:= SIZEOF(BYTE);
M_BuildUINT8.aMessage[1] 	:= nInValue;
END_METHOD

END_FUNCTION_BLOCK

// ---- KNXnetIPTunnelingServer/POUs/KNX_DatapointTypes_Interpreter.TcPOU
(*
:Description: function block for interpret the DPT from KNX devices
:Instructions for use: instantiate this function block to use the implemented interface I_KNX_DPT_Interpreter and its methods to interpret the KNX messages correctly
*)
FUNCTION_BLOCK KNX_DatapointTypes_Interpreter IMPLEMENTS I_KNX_DPT_Interpreter

METHOD M_InterpretAs2Bit : ST_KNX_DPT_B2
VAR_IN_OUT
	aInData		: ARRAY[*] OF BYTE;
END_VAR
M_InterpretAs2Bit.bBit1 := aInData[LOWER_BOUND(aInData,1)].0;
M_InterpretAs2Bit.bBit2 := aInData[LOWER_BOUND(aInData,1)].1;
END_METHOD

METHOD M_InterpretAsBool : BOOL
VAR_IN_OUT
	aInData		: ARRAY[*] OF BYTE;
END_VAR
M_InterpretAsBool := BYTE_TO_BOOL(aInData[LOWER_BOUND(aInData,1)]);
END_METHOD

METHOD M_InterpretAsDimming : ST_KNX_DPT_ControlDimming
VAR_IN_OUT
	aInData		: ARRAY[*] OF BYTE;
END_VAR
M_InterpretAsDimming.bControl 	:= aInData[LOWER_BOUND(aInData,1)].3;
M_InterpretAsDimming.nStepCode	:= aInData[LOWER_BOUND(aInData,1)] AND 16#07;
END_METHOD

METHOD M_InterpretAsFloat16 : REAL
VAR_IN_OUT
	aInData		: ARRAY[*] OF BYTE;
END_VAR
VAR
	nMantissa		: WORD;
	nSignMantissa	: INT;
	//nExponent		: INT;
	fFloat			: REAL;
	//nSign			: INT;
	
	
	
	nExponent		: WORD;
	nSign			: INT;
	fMAXValue		: REAL;
	nValue			: INT;
	nResult			: WORD;
END_VAR
//nSign 			:= BIT_TO_INT(stInData[LOWER_BOUND(stInData,1)].7);
//nMantissa 		:= SHL(BYTE_TO_WORD(stInData[LOWER_BOUND(stInData,1)]) AND 16#07, 8);
//nMantissa 		:= nMantissa OR BYTE_TO_WORD(stInData[LOWER_BOUND(stInData,1) + 1]);
//nSignMantissa 	:= WORD_TO_INT(nMantissa);
//IF nSign = 1 THEN
//	// negative value
//	nMantissa := NOT nMantissa;
//	nMantissa := nMantissa OR (NOT 16#F800);
//	nSignMantissa := WORD_TO_INT(nMantissa + 1);
//	nSignMantissa := nSignMantissa * -1;
//END_IF
//nExponent := BYTE_TO_INT(stInData[LOWER_BOUND(stInData,1)] AND 16#78);
//M_InterpretAsFloat16 := LREAL_TO_REAL(0.01 * nSignMantissa * EXPT(2, nExponent));


nResult := SHL(BYTE_TO_WORD(aInData[LOWER_BOUND(aInData,1)]), 8);
nResult := nResult OR BYTE_TO_WORD(aInData[LOWER_BOUND(aInData,1)+1]);


	IF nResult/2048<16 THEN
		nSign:=1;
		nExponent:=nResult/2048;
	ELSE
		nSign:=-1;
		nExponent:=(nResult/2048)-16;
	END_IF
	fMAXValue:=LREAL_TO_REAL(EXPT(2,nExponent)*20.48);
	
	nValue:=UINT_TO_INT(nResult MOD 2048);
	IF nSign<0 THEN
		nValue := 2048-nValue;
	END_IF
	M_InterpretAsFloat16:=(INT_TO_REAL(nValue)/2048)*fMAXValue*nSign;
END_METHOD

METHOD M_InterpretAsFloat32 : Real
VAR_IN_OUT
	aInData		: ARRAY[*] OF BYTE;
END_VAR
VAR
	
	nWord			: DWORD;
	pReal			: POINTER TO REAL;
	i				: INT;
END_VAR
FOR i := 0 TO 3 DO
	nWord:=nWord + SHL(aInData[4-i],i*8);
END_FOR

pReal := ADR(nWord);
M_InterpretAsFloat32 := pReal^;
END_METHOD

METHOD M_InterpretAsINT16 : INT
VAR_IN_OUT
	aInData		: ARRAY[*] OF BYTE;
END_VAR
VAR
	nResult			: WORD;
END_VAR
nResult := SHL(BYTE_TO_WORD(aInData[LOWER_BOUND(aInData,1)]), 8);
nResult := nResult OR BYTE_TO_WORD(aInData[LOWER_BOUND(aInData,1)+1]);
M_InterpretAsINT16 := WORD_TO_INT(nResult);
END_METHOD

METHOD M_InterpretAsINT32 : DINT
VAR_IN_OUT
	aInData		: ARRAY[*] OF BYTE;
END_VAR
VAR
	nResult			: DWORD;
END_VAR
nResult := SHL(BYTE_TO_DWORD(aInData[LOWER_BOUND(aInData,1)]), 8*3);
nResult := nResult OR SHL(BYTE_TO_DWORD(aInData[LOWER_BOUND(aInData,1)+1]), 8*2);
nResult := nResult OR SHL(BYTE_TO_DWORD(aInData[LOWER_BOUND(aInData,1)+2]), 8);
nResult := nResult OR BYTE_TO_DWORD(aInData[LOWER_BOUND(aInData,1)+3]);
M_InterpretAsINT32 := DWORD_TO_DINT(nResult);
END_METHOD

METHOD M_InterpretAsUINT16 : UINT
VAR_IN_OUT
	aInData		: ARRAY[*] OF BYTE;
END_VAR
VAR
	nResult			: UINT;
END_VAR
nResult := SHL(BYTE_TO_WORD(aInData[LOWER_BOUND(aInData,1)]),8);
nResult := nResult OR BYTE_TO_WORD(aInData[LOWER_BOUND(aInData,1)+1]);
M_InterpretAsUINT16 := nResult;
END_METHOD

METHOD M_InterpretAsUINT32 : UDINT
VAR_IN_OUT
	aInData		: ARRAY[*] OF BYTE;
END_VAR
VAR
	nResult			: UDINT;
END_VAR
nResult := SHL(BYTE_TO_DWORD(aInData[LOWER_BOUND(aInData,1)]),8*3);
nResult := nResult OR SHL(BYTE_TO_DWORD(aInData[LOWER_BOUND(aInData,1)]+1),8*2);
nResult := nResult OR SHL(BYTE_TO_DWORD(aInData[LOWER_BOUND(aInData,1)]+2),8);
nResult := nResult OR BYTE_TO_DWORD(aInData[LOWER_BOUND(aInData,1)]+3);
M_InterpretAsUINT32 := nResult;
END_METHOD

METHOD M_InterpretAsUINT8 : BYTE
VAR_IN_OUT
	aInData		: ARRAY[*] OF BYTE;
END_VAR
M_InterpretAsUINT8 := aInData[LOWER_BOUND(aInData,1)];
END_METHOD

METHOD M_InterpretNewMessage : BOOL
VAR_IN_OUT
	bInData		: BOOL;
END_VAR
M_InterpretNewMessage := bInData;
END_METHOD

END_FUNCTION_BLOCK

// ---- KNXnetIP_Devices/Button/FB_KNXnetIP_Button.TcPOU
(*
:Description: device function block for a normal button, it will interpret the button state as bool
*)
FUNCTION_BLOCK FB_KNXnetIP_Button EXTENDS FB_KNXnetIP_Device_Abstract
VAR_INPUT
	bInToggle			: BOOL := FALSE;			// activate toggle with high rising edge
	tInLongPressedTime	: TIME := T#0S;				// not used if not parameterized or Time = Os
END_VAR
VAR_OUTPUT
	bOutState			: BOOL;						// state of output
	bOutLongPressed		: BOOL;						// button long pressed
	bOutRunning			: BOOL;						// function block is working correctly
END_VAR                             				
VAR
	bBtnState			: BOOL;
	rtBtnState			: R_TRIG;
END_VAR
VAR PERSISTENT                      				
	bLastState			: BOOL;						// stored last state of input
END_VAR

IF ipInKnxTunneling = 0 OR ipInKnxInterpreter = 0 OR NOT ipInKnxTunneling.P_G_IsConnected THEN
	bOutState := bLastState;
	RETURN;
END_IF
bOutRunning := TRUE;
bBtnState 	:= ipInKnxInterpreter.M_InterpretAsBool(ipInKnxTunneling.P_G_GroupAddressMessages.aMessage[stInKnxGroupAddress.nFirst, stInKnxGroupAddress.nMiddle, stInKnxGroupAddress.nLow]);
IF NOT bInToggle THEN
	bOutState := bBtnState;
ELSE
	rtBtnState(CLK := bBtnState);
	IF rtBtnState.Q THEN
		bOutState := NOT bOutState;
	END_IF
END_IF
bLastState 		:= bOutState;
bOutLongPressed	:= M_LongPressed();

METHOD PRIVATE M_LongPressed : BOOL
VAR_INST
	tnLongPressed		: TON;
END_VAR
VAR CONSTANT
	ctLongPressed		: TIME := T#1S;				// long pressed time
END_VAR
IF tInLongPressedTime = T#0S THEN
	tnLongPressed(IN := bBtnState, PT := ctLongPressed);
ELSE	
	tnLongPressed(IN := bBtnState, PT := tInLongPressedTime);
END_IF
M_LongPressed := tnLongPressed.Q;
END_METHOD

END_FUNCTION_BLOCK

// ---- KNXnetIP_Devices/FB_KNXnetIP_Device_Abstract.TcPOU
FUNCTION_BLOCK ABSTRACT FB_KNXnetIP_Device_Abstract
VAR_INPUT
	stInKnxGroupAddress		: ST_KNX_GroupAddress;
	ipInKnxTunneling		: I_KNXnetIP_Tunneling;
	ipInKnxInterpreter		: I_KNX_DPT_Interpreter;
	ipInKnxBuilder			: I_KNX_DPT_Builder;
END_VAR

END_FUNCTION_BLOCK

// ---- KNXnetIP_Devices/Light/FB_KNXnetIP_Light.TcPOU
(*
:Description: device function block for a normal light, it will send the state as bool
*)
FUNCTION_BLOCK FB_KNXnetIP_Light EXTENDS FB_KNXnetIP_Device_Abstract
VAR_INPUT
	bInOnOff			: BOOL;		// light is ON (TRUE) or OFF (FALSE)
END_VAR
VAR_OUTPUT
	bOutRunning			: BOOL;		// function block is working correctly
END_VAR
VAR
	rtConnected			: R_TRIG;	// rising trigger of connected state
END_VAR
VAR PERSISTENT
	bLastState			: BOOL;		// stored last state of input
END_VAR

IF ipInKnxTunneling = 0 OR ipInKnxBuilder = 0 OR NOT ipInKnxTunneling.P_G_IsConnected THEN
	RETURN;
END_IF
bOutRunning := TRUE;
rtConnected(CLK := ipInKnxTunneling.P_G_IsConnected);	// send message if connection is valid
IF bInOnOff <> bLastState THEN //OR rtConnected.Q THEN
	bLastState := bInOnOff;
	ipInKnxTunneling.M_TransmitMessage(stInKnxGroupAddress, ipInKnxBuilder.M_BuildBool(bInOnOff));
END_IF

END_FUNCTION_BLOCK

// ---- Project Information/F_GetCompany.TcPOU
// This function has been automatically generated from the project information.
{attribute 'signature_flag' := '1073741824'}
{attribute 'TcGenerated'}
{attribute 'no-analysis'}
FUNCTION F_GetCompany : WSTRING
VAR_INPUT
	
END_VAR

F_GetCompany := "Gauggel";

END_FUNCTION

// ---- Project Information/F_GetTitle.TcPOU
// This function has been automatically generated from the project information.
{attribute 'signature_flag' := '1073741824'}
{attribute 'TcGenerated'}
{attribute 'no-analysis'}
FUNCTION F_GetTitle : WSTRING
VAR_INPUT
	
END_VAR

F_GetTitle := "TcKNXnetIP_Tunneling_Lib";

END_FUNCTION

// ---- Project Information/F_GetVersion.TcPOU
// This function has been automatically generated from the project information.
{attribute 'signature_flag' := '1073741824'}
{attribute 'TcGenerated'}
{attribute 'no-analysis'}
FUNCTION F_GetVersion : ST_LibVersion
VAR_INPUT
	
END_VAR

F_GetVersion.iMajor := 1;
F_GetVersion.iMinor := 0;
F_GetVersion.iBuild := 0;
F_GetVersion.iRevision := 0;
F_GetVersion.sVersion := '1.0.0';
F_GetVersion.nFlags := 1;

END_FUNCTION
